Yaskawa INFORM job: OK_R2_O57-69(1)(90,0)OLD.JBI

/JOB
//NAME OK_R2_O57-69(1)(90,0)OLD
//POS
///NPOS 677,677,677,19,0,0
///TOOL 0
///POSTYPE PULSE
///PULSE
C00000=-115282,71817,32941,48127,54711,-22306
C00001=-113844,78377,40832,48113,52960,-22533
C00002=-113286,81152,44222,48167,52223,-22657
C00003=-112658,81907,45149,47913,51773,-22558
C00004=-113286,81152,44222,48167,52223,-22657
C00005=-114841,82290,45172,49039,53033,-23084
C00006=-115003,85006,48527,49507,52672,-23414
C00007=-114841,82290,45172,49039,53033,-23084
C00008=-115410,79539,41800,48987,53774,-22957
C00009=-116878,73048,33960,49005,55537,-22725
C00010=-114631,73287,21777,30026,68466,-13972
C00011=-107687,96017,31887,4043,95712,-4008
C00012=-107423,99778,39901,3942,92708,-4025
C00013=-107321,101469,43344,3906,91457,-4032
C00014=-107321,100752,43692,3904,90875,-4050
C00015=-107321,101469,43344,3906,91457,-4032
C00016=-107333,102312,44062,3909,91449,-4036
C00017=-107226,104962,47560,3875,90654,-4028
C00018=-107333,102312,44062,3909,91449,-4036
C00019=-107436,100611,40601,3946,92706,-4028
C00020=-107700,96832,32553,4047,95722,-4011
C00021=-108294,85696,32273,9932,91830,-10529
C00022=-107637,89717,40349,9733,88894,-10552
C00023=-107381,91513,43820,9663,87669,-10565
C00024=-107382,91052,44496,9665,87024,-10615
C00025=-107381,91513,43820,9663,87669,-10565
C00026=-107317,92116,44380,9645,87627,-10547
C00027=-107050,94613,47567,9574,86928,-10515
C00028=-107317,92116,44380,9645,87627,-10547
C00029=-107572,90309,40892,9715,88857,-10534
C00030=-108227,86267,32782,9914,91803,-10510
C00031=-112253,73171,16618,11071,95439,-11452
C00032=-122495,9844,5157,25727,54942,-17539
C00033=-121156,16110,12600,25480,53295,-17364
C00034=-120642,18694,15712,25408,52605,-17310
C00035=-120643,19132,17389,25673,51873,-17507
C00036=-120642,18694,15712,25408,52605,-17310
C00037=-120849,18005,15099,25505,52689,-17383
C00038=-120429,19971,16941,25331,52448,-17252
C00039=-120849,18005,15099,25505,52689,-17383
C00040=-121367,15431,12007,25581,53375,-17439
C00041=-122717,9186,4605,25835,55013,-17621
C00042=-138494,21467,-20962,-13510,88545,-918
C00043=-172227,55679,50190,-52098,32064,25809
C00044=-172226,58151,57267,-56252,30204,27980
C00045=-172259,73719,75605,-61261,28412,30549
C00046=-172259,73719,75605,-61261,28412,30549
C00047=-172291,75568,77861,-61964,28174,30905
C00048=-172279,67127,67655,-59517,29872,29717
C00049=-172279,67127,67655,-59517,29872,29717
C00050=-172707,68806,69649,-59823,29417,29854
C00051=-172279,67127,67655,-59517,29872,29717
C00052=-172484,58153,57400,-56260,30062,27978
C00053=-173076,56772,55516,-55150,29916,27380
C00054=-172487,71730,32634,-35509,46109,16330
C00055=-172505,79305,41756,-36484,44696,16958
C00056=-171934,80372,43058,-38467,45492,17923
C00057=-171699,86165,50208,-39533,44475,18576
C00058=-171934,80372,43058,-38467,45492,17923
C00059=-171934,80372,43058,-38467,45492,17923
C00060=-171934,80372,43058,-38467,45492,17923
C00061=-171934,80372,43058,-38467,45492,17923
C00062=-171934,80372,43058,-38467,45492,17923
C00063=-172992,69880,30345,-34862,46288,15983
C00064=-172199,59331,16615,-33939,49113,15228
C00065=-172399,68292,26984,-34663,47555,15757
C00066=-172399,68292,26984,-34663,47555,15757
C00067=-172079,70977,30156,-35213,47204,16071
C00068=-172399,68292,26984,-34663,47555,15757
C00069=-172399,68292,26984,-34663,47555,15757
C00070=-173084,68902,27700,-34193,47184,15559
C00071=-172399,68292,26984,-34663,47555,15757
C00072=-172399,68292,26984,-34663,47555,15757
C00073=-173171,57722,14227,-32886,49296,14681
C00074=-136545,44574,15947,-43124,46451,20365
C00075=-172050,-124043,-93312,-19428,16171,9287
C00076=-155648,-70131,-83120,13924,61027,17443
C00077=-136290,-23516,-60153,14090,83188,29885
C00078=-136350,-23051,-59906,14078,83550,29899
C00079=-136350,-23664,-59049,14098,82729,29803
C00080=-136350,-23051,-59906,14078,83550,29899
C00081=-134790,5262,-45049,12672,103577,12599
C00082=-134622,7343,-43237,12633,103510,12643
C00083=-134790,5262,-45049,12672,103577,12599
C00084=-130650,-5709,-52245,4545,96168,15148
C00085=-131657,-5407,-52003,4830,96225,14850
C00086=-130650,-5709,-52245,4545,96168,15148
C00087=-132561,-6063,-53863,7723,97717,11875
C00088=-132436,-8720,-59337,7740,99694,12036
C00089=-132445,-1782,-62924,7952,105415,12403
C00090=-141601,37323,-23290,10329,102010,9516
C00091=-93172,55874,9388,-1843,94357,23900
C00092=-93485,56784,11787,-1769,93341,23816
C00093=-93485,56329,12545,-1767,92641,23826
C00094=-93485,56784,11787,-1769,93341,23816
C00095=-93464,57012,11403,-1775,93695,23818
C00096=-93714,59095,13766,-1718,93307,23745
C00097=-93464,57012,11403,-1775,93695,23818
C00098=-94351,55649,10247,-1575,93690,23540
C00099=-95033,54913,9421,-1421,93808,23324
C00100=-94351,55649,10247,-1575,93690,23540
C00101=-94041,54751,7862,-1648,94701,23624
C00102=-93250,52756,2164,-1838,97197,23834
C00103=-93258,57323,-1415,-1867,101744,23764
C00104=-108708,74058,35602,41753,92549,11625
C00105=-107609,77867,43172,41468,89995,11080
C00106=-107179,79572,46434,41382,88936,10847
C00107=-107179,79487,47575,41378,88368,10623
C00108=-107179,79572,46434,41382,88936,10847
C00109=-85041,17756,-8276,-11251,50625,9461
C00110=-85416,19690,-6470,-10982,50459,9320
C00111=-85041,17756,-8276,-11251,50625,9461
C00112=-87036,75660,30192,-3211,91902,25887
C00113=-87645,74633,28952,-3076,92115,25688
C00114=-87036,75660,30192,-3211,91902,25887
C00115=-86708,74680,27642,-3289,92979,25963
C00116=-85872,72543,21626,-3493,95611,26155
C00117=-85876,74587,19798,-3512,97782,26092
C00118=-86821,26768,-33196,-3418,105774,25582
C00119=-56288,-65443,-100505,-9939,102051,34984
C00120=-94872,-76247,-37251,-15619,10327,-42827
C00121=-113351,-68967,-59155,816,27582,-73246
C00122=-112415,-66495,-57032,-529,27544,-72574
C00123=-112416,-66088,-55565,-540,26850,-72568
C00124=-112415,-66495,-57032,-529,27544,-72574
C00125=-125946,-59954,-52375,33832,33505,-67413
C00126=-125801,-56324,-50419,33152,34009,-67051
C00127=-125986,-60936,-52893,34026,33366,-67517
C00128=-133343,-54797,-49167,48338,43724,-75418
C00129=-132401,-55055,-49311,47843,43188,-75129
C00130=-125164,-63316,-53721,33839,32440,-67422
C00131=-126284,-65474,-55722,34821,32994,-67941
C00132=-120687,-90156,-48971,65843,10407,33929
C00133=-163424,-29173,-12092,69684,68620,47205
C00134=-170503,-20236,-5842,69401,73657,46605
C00135=-165190,-726,9323,69215,70349,47621
C00136=-177502,-61167,-55570,67933,81710,43621
C00137=-170775,-70491,-60275,67726,76450,43734
C00138=-168988,-72616,-61292,67687,75067,43782
C00139=-168256,-73449,-61686,67672,74502,43804
C00140=-168255,-73403,-61547,67686,74477,43777
C00141=-168256,-73449,-61686,67672,74502,43804
C00142=-168129,-73592,-61753,67670,74405,43808
C00143=-166480,-73871,-61885,67549,73279,44015
C00144=-168129,-73592,-61753,67670,74405,43808
C00145=-168863,-72760,-61361,67684,74971,43786
C00146=-170655,-70639,-60347,67723,76357,43737
C00147=-176850,-62168,-56094,67907,81198,43629
C00148=-197320,-70186,-60126,68463,94301,40195
C00149=-181036,-69697,-66198,61349,79658,32659
C00150=-200540,-66438,-67217,63628,100285,-15829
C00151=-127293,-88890,-117674,21964,112183,-47373
C00152=-127884,-113870,-117586,20406,100261,-49782
C00153=-127000,-93154,-82052,19489,96345,-50169
C00154=-123343,-94047,-79271,19637,93420,-49322
C00155=-121848,-94244,-78089,19702,92278,-48969
C00156=-121839,-92557,-75577,19688,91637,-49071
C00157=-121848,-94244,-78089,19702,92278,-48969
C00158=-119969,-93354,-78147,19815,92288,-48290
C00159=-118624,-93308,-78129,19884,91973,-47856
C00160=-119969,-93354,-78147,19815,92288,-48290
C00161=-121462,-93189,-79339,19761,93422,-48643
C00162=-125120,-92380,-82146,19635,96326,-49491
C00163=-116413,-89407,-85315,-11170,94586,69972
C00164=-118284,-91858,-82643,-11111,91478,69605
C00165=-119058,-92674,-81496,-11095,90266,69446
C00166=-119076,-90876,-79147,-11092,89752,69486
C00167=-119058,-92674,-81496,-11095,90266,69446
C00168=-118796,-98042,-83265,-11090,88662,69679
C00169=-118779,-98894,-83439,-11090,88340,69713
C00170=-118796,-98042,-83265,-11090,88662,69679
C00171=-123354,-93602,-81963,-11047,89491,68033
C00172=-124901,-93499,-81921,-11022,89307,67516
C00173=-123354,-93602,-81963,-11047,89491,68033
C00174=-122534,-92869,-83147,-11066,90689,68210
C00175=-120547,-90622,-85912,-11132,93767,68620
C00176=-120571,-90661,-98380,-11386,101275,67925
C00177=-125069,-105236,-119201,46912,96955,7142
C00178=-121279,-99548,-114464,46207,95099,8000
C00179=-119841,-97303,-112552,45921,94382,8319
C00180=-119848,-96543,-111162,45886,94057,8165
C00181=-119841,-97303,-112552,45921,94382,8319
C00182=-121259,-87971,-110760,46601,97668,9229
C00183=-121257,-87068,-110229,46617,97763,9276
C00184=-121259,-87971,-110760,46601,97668,9229
C00185=-122654,-89805,-112582,46929,98462,8982
C00186=-126320,-94321,-117059,47765,100534,8329
C00187=-125132,-111985,-108710,18887,62200,-22139
C00188=-122150,-102499,-103347,17190,63051,-20837
C00189=-121052,-98905,-101202,16573,63333,-20372
C00190=-121051,-97796,-99654,16626,62964,-20427
C00191=-121052,-98905,-101202,16573,63333,-20372
C00192=-120662,-97381,-100799,16308,63770,-20159
C00193=-118649,-97310,-100773,15302,63405,-19446
C00194=-120662,-97381,-100799,16308,63770,-20159
C00195=-120717,-96579,-100674,16290,64103,-20131
C00196=-120723,-93199,-99767,16143,65237,-19969
C00197=-120717,-96579,-100674,16290,64103,-20131
C00198=-121791,-100117,-102825,16885,63842,-20577
C00199=-124704,-109452,-108202,18522,63043,-21827
C00200=-114740,-109793,-107699,-22238,66313,27441
C00201=-118303,-101714,-102676,-20552,66389,26052
C00202=-119630,-98598,-100655,-19919,66404,25543
C00203=-119639,-97485,-99100,-19970,66039,25605
C00204=-119630,-98598,-100655,-19919,66404,25543
C00205=-121461,-98371,-100392,-19110,65937,24929
C00206=-122362,-98343,-100381,-18703,65740,24620
C00207=-120869,-98346,-100801,-19339,66320,25087
C00208=-120753,-95574,-99975,-19267,67213,24978
C00209=-120759,-92226,-99069,-19116,68313,24791
C00210=-120753,-95574,-99975,-19267,67213,24978
C00211=-119475,-98647,-102011,-19875,67204,25461
C00212=-116042,-106621,-107071,-21497,67130,26779
C00213=-113894,-113482,-108593,-25442,60982,30098
C00214=-117729,-104898,-103745,-23262,61171,28471
C00215=-119152,-101582,-101788,-22448,61245,27877
C00216=-119170,-99952,-99576,-22546,60754,27973
C00217=-119152,-101582,-101788,-22448,61245,27877
C00218=-121013,-102333,-103012,-21430,61098,27156
C00219=-123141,-102270,-102988,-20324,60582,26401
C00220=-121013,-102333,-103012,-21430,61098,27156
C00221=-120862,-89775,-98642,-20835,64658,26523
C00222=-120866,-85397,-96829,-20654,65721,26323
C00223=-120862,-89775,-98642,-20835,64658,26523
C00224=-119577,-92842,-100627,-21537,64647,27018
C00225=-116128,-100765,-105545,-23412,64594,28369
C00226=-120616,-96668,-103675,-23957,64374,45643
C00227=-120616,-97077,-101536,-24254,62975,45956
C00228=-120353,-97213,-100348,-24551,62319,46212
C00229=-118869,-97129,-100639,-25236,62958,46664
C00230=-120614,-98300,-102259,-24293,62807,45995
C00231=-123308,-94059,-109732,-20810,92119,41464
C00232=-120560,-97114,-101199,-23431,86244,43216
C00233=-120636,-92458,-99001,-23404,87178,43005
C00234=-120616,-97068,-101477,-23418,86408,43164
C00235=-120616,-96536,-104145,-23405,88172,42819
C00236=-120615,-97089,-97846,-24331,46439,48575
C00237=-120614,-96205,-89198,-26458,42021,49913
C00238=-120613,-95813,-87227,-26966,41113,50220
C00239=-120147,-95634,-86429,-27555,40908,50556
C00240=-118868,-95589,-86413,-28580,41350,51125
C00241=-120611,-96965,-88121,-26990,41076,50233
C00242=-120469,-95981,-105264,-23437,89109,42688
C00243=-120355,-96765,-101896,-23463,86860,43169
C00244=-119463,-95970,-102962,-19996,114254,37918
C00245=-120616,-96568,-103294,-18987,119739,36439
C00246=-120617,-95735,-106079,-19458,121767,36056
C00247=-120683,-72727,-118704,-1403,106780,1205
C00248=-120616,-97110,-101484,23732,56591,-46685
C00249=-120615,-97329,-97421,24453,54195,-47265
C00250=-120615,-97216,-95276,24833,53043,-47558
C00251=-120317,-97140,-94459,24795,52533,-47555
C00252=-120613,-98372,-96050,24869,52935,-47585
C00253=-122362,-97116,-94396,26052,53130,-48332
C00254=-120517,-95602,-107135,23321,90071,-42137
C00255=-120393,-96024,-106061,23287,89229,-42258
C00256=-120510,-96280,-105304,23307,88709,-42400
C00257=-120617,-95942,-106325,23333,89477,-42288
C00258=-120617,-94838,-108784,23367,91395,-41914
C00259=-120619,-89077,-114974,23678,97628,-40680
C00260=-119375,-87803,-114046,-9627,73434,-76892
C00261=-119874,-91001,-111320,-9540,70103,-76790
C00262=-120074,-92022,-110137,-9508,68845,-76756
C00263=-120388,-88035,-108953,-9268,70114,-76963
C00264=-120068,-92699,-111595,-9479,69387,-76797
C00265=-120617,-92323,-109789,-9348,67950,-76861
C00266=-120617,-92636,-109412,-9435,67087,-76774
C00267=-120617,-92966,-108935,-9385,65680,-76698
C00268=-120617,-93485,-108112,-8702,63167,-76584
C00269=-120617,-93807,-107566,-7310,61334,-76551
C00270=-120617,-93899,-107425,-5913,60596,-76588
C00271=-120617,-91887,-110532,-5160,63404,-76609
C00272=-120617,-91830,-110616,-4244,63440,-76636
C00273=-120617,-91600,-110911,-2665,64017,-76695
C00274=-120618,-91126,-111456,-1065,65432,-76762
C00275=-120618,-90436,-112164,126,67515,-76814
C00276=-120618,-89799,-112749,669,69377,-76843
C00277=-120618,-88579,-113586,734,71430,-76721
C00278=-120618,-87737,-114188,674,73665,-76767
C00279=-120618,-86710,-114840,-40,76341,-76871
C00280=-120619,-85981,-115253,-1370,78289,-77032
C00281=-120619,-85769,-115356,-2649,79041,-77176
C00282=-118258,-89310,-112812,-4565,75923,-76275
C00283=-117029,-89279,-112689,-5985,75998,-75947
C00284=-115084,-89307,-112300,-8369,75681,-75412
C00285=-113300,-89514,-111627,-10775,74614,-74872
C00286=-112191,-89952,-110802,-12600,72842,-74453
C00287=-112162,-90329,-110382,-13115,71673,-74372
C00288=-116808,-91534,-110372,-11031,70029,-75758
C00289=-120074,-92022,-110137,-9508,68845,-76756
C00290=-119874,-91001,-111320,-9540,70103,-76790
C00291=-119375,-87803,-114046,-9627,73434,-76892
C00292=-120613,-96141,-86612,-20456,81391,53018
C00293=-120613,-95201,-83022,-20541,79769,53295
C00294=-121508,-95240,-81659,-19950,77874,52000
C00295=-119108,-93506,-81277,-20755,79958,53812
C00296=-120703,-96226,-83293,-20548,79408,53324
C00297=-120206,-95185,-82888,-16285,85651,57184
C00298=-120275,-93619,-78099,-16321,83579,57434
C00299=-120502,-93714,-78663,-14162,87512,64436
C00300=-120613,-94474,-80645,-13297,90613,68078
C00301=-120613,-95649,-84682,-13324,92446,67881
C00302=-120615,-97441,-93706,-13451,96957,67391
C00303=-117944,-114132,-91182,23549,57658,-33742
C00304=-120612,-94052,-79174,30375,49115,-27391
C00305=-120612,-92306,-74262,31338,47277,-28046
C00306=-120611,-91624,-72518,31687,46656,-28277
C00307=-120558,-89719,-71004,31635,46677,-28249
C00308=-120609,-92783,-73582,31657,46706,-28257
C00309=-122365,-91326,-71808,32798,47083,-29054
C00310=-121100,-96285,-86968,23801,78483,-44635
C00311=-121303,-91870,-73161,24426,72832,-45883
C00312=-121523,-93334,-74795,23462,83796,-58035
C00313=-120612,-93040,-76284,23523,87550,-60648
C00314=-120612,-94304,-79928,23524,89017,-60360
C00315=-192979,-49879,-84133,31949,90821,-59300
C00316=-226136,-49296,-77583,43048,96139,-60221
C00317=-194231,-43574,-37464,64429,96533,35524
C00318=-168190,-921,2356,69742,86936,65420
C00319=-157686,-14873,-8721,69811,79682,66593
C00320=-155170,-17431,-10634,69793,77924,66853
C00321=-154140,-18406,-11354,69782,77205,66960
C00322=-154960,-19735,-12328,69815,77730,66818
C00323=-154139,-18877,-12975,69638,77486,67291
C00324=-152416,-19959,-12491,68149,70274,62953
C00325=-151462,-20771,-13080,67326,65877,57651
C00326=-150584,-21490,-13598,66880,61935,51327
C00327=-149448,-22378,-14235,66195,57985,45258
C00328=-150364,-21665,-13724,66599,59939,44567
C00329=-146294,-24621,-15825,64622,49633,44461
C00330=-147024,-24129,-15478,65026,50858,44122
C00331=-148183,-23314,-14902,65711,53127,43519
C00332=-150746,-21357,-13503,66515,56405,42739
C00333=-151844,-20450,-12847,67017,58691,42205
C00334=-154160,-18394,-11345,67568,61790,41547
C00335=-155150,-17454,-10651,67918,63984,41080
C00336=-156307,-16307,-9798,68285,66690,40524
C00337=-158578,-13896,-7981,68632,70174,39857
C00338=-158236,-14274,-8267,68563,69306,40027
C00339=-158768,-13688,-7823,68593,69674,39964
C00340=-160083,-12191,-6676,68663,70584,39811
C00341=-163356,-38025,-17867,70039,68206,46757
C00342=-171321,-47804,-23743,70196,73038,45095
C00343=-120855,-117042,-83065,287,50429,-281
C00344=-120852,-56541,-79529,233,79340,-219
C00345=-120696,51333,26745,175,69370,-180
C00346=-120686,107948,75662,172,68359,-178
C00347=-120686,108277,78684,174,66668,-180
C00348=-120673,108876,79912,172,66223,-177
C00349=-120685,108330,78544,174,66782,-180
C00350=-120704,104314,74519,181,67195,-186
C00351=-120673,108876,79912,172,66223,-177
C00352=-121521,109835,81177,5465,66399,-4971
C00353=-123474,116640,90211,14625,67368,-13734
C00354=-120128,113257,88761,29498,73318,-26772
C00355=-120686,108838,82574,29428,74862,-26590
C00356=-121763,107966,77633,29394,77512,-26324
C00357=-120686,107962,76375,6322,66410,-5366
C00358=-120686,108055,77304,6346,65890,-5395
C00359=-117369,97126,64252,10958,70846,-6903
C00360=-120686,108293,79018,6392,64962,-5445
C00361=-120992,104893,75799,6510,65219,-5544
C00362=-117369,97126,64252,10958,70846,-6903
C00363=-120630,108400,78956,19693,72345,-15662
C00364=-120761,107752,79258,26649,76197,-23334
C00365=-121775,107524,77536,26798,77367,-23449
C00366=-120025,79294,29666,22432,87187,-16596
C00367=-146832,96040,51096,-31563,98712,41471
C00368=-156862,88199,54516,-55770,96758,71489
C00369=-156858,88352,61458,-55305,94312,73083
C00370=-157852,91445,67330,-55099,92539,73648
C00371=-158245,92835,69884,-55033,91801,73892
C00372=-157951,96204,74186,-54996,91433,74294
C00373=-157784,91273,67188,-55102,92578,73662
C00374=-158040,92399,69988,-55026,91755,74041
C00375=-159291,95627,71523,-51291,93332,81554
C00376=-160209,98279,73182,-48482,94322,83905
C00377=-159956,97162,70645,-48575,95125,83623
C00378=-159321,94794,64867,-48849,97041,82959
C00379=-174197,80542,71118,-15802,102714,62389
C00380=-174195,80556,71135,-15802,102711,62390
C00381=-174195,80561,71142,-15801,102710,62390
C00382=-173773,83477,74756,-15654,102092,62625
C00383=-174194,79765,68888,-15876,103653,62265
C00384=-174199,80535,71109,-11568,105990,64366
C00385=-174198,80539,71114,-12074,105866,67869
C00386=-174201,80518,71089,-8660,108894,72599
C00387=-174202,80510,71078,-8661,108896,72599
C00388=-174205,80488,71052,-8662,108901,72597
C00389=-174210,80448,71002,-8664,108910,72595
C00390=-160796,99181,68474,-21491,79626,-54117
C00391=-160795,99200,68498,-21491,79622,-54116
C00392=-160795,99207,68507,-21491,79620,-54116
C00393=-160747,98987,66984,-21457,80402,-54239
C00394=-161332,101028,70752,-21395,79065,-54211
C00395=-160795,99207,68507,-21491,79620,-54116
C00396=-160795,99200,68498,-21491,79622,-54116
C00397=-160796,99181,68474,-21491,79626,-54117
C00398=-156887,88424,61529,-55303,94292,73080
C00399=-157880,91522,67408,-55097,92517,73646
C00400=-158273,92915,69967,-55032,91779,73890
C00401=-157979,96289,74274,-54994,91410,74293
C00402=-157812,91350,67266,-55100,92556,73660
C00403=-158068,92478,70069,-55024,91733,74039
C00404=-159318,95712,71612,-51289,93309,81552
C00405=-160236,98368,73278,-48480,94299,83903
C00406=-159983,97249,70737,-48574,95102,83621
C00407=-159349,94875,64951,-48847,97020,82956
C00408=-174197,80542,71118,-15802,102714,62389
C00409=-174195,80555,71135,-15802,102711,62390
C00410=-174195,80561,71141,-15801,102710,62390
C00411=-173773,83477,74755,-15654,102093,62624
C00412=-174194,79764,68887,-15876,103653,62265
C00413=-174199,80534,71109,-11568,105990,64366
C00414=-174198,80538,71114,-12074,105866,67869
C00415=-174201,80518,71088,-8660,108894,72599
C00416=-174202,80509,71078,-8661,108896,72599
C00417=-174205,80488,71051,-8662,108901,72597
C00418=-174210,80448,71002,-8664,108910,72595
C00419=-160796,99181,68473,-21491,79626,-54117
C00420=-160795,99199,68497,-21491,79622,-54116
C00421=-160795,99206,68506,-21491,79620,-54116
C00422=-160747,98986,66983,-21457,80402,-54239
C00423=-161332,101028,70752,-21395,79065,-54211
C00424=-160795,99206,68506,-21491,79620,-54116
C00425=-160795,99199,68497,-21491,79622,-54116
C00426=-160796,99181,68473,-21491,79626,-54117
C00427=-156915,88496,61599,-55301,94271,73077
C00428=-157907,91600,67487,-55096,92496,73644
C00429=-158301,92995,70050,-55030,91757,73888
C00430=-158006,96373,74363,-54993,91387,74291
C00431=-157840,91427,67345,-55098,92535,73658
C00432=-158096,92558,70151,-55023,91711,74037
C00433=-159346,95797,71702,-51288,93287,81550
C00434=-160263,98458,73375,-48479,94275,83902
C00435=-160010,97336,70829,-48572,95080,83619
C00436=-159376,94956,65035,-48845,96998,82954
C00437=-174197,80541,71117,-15802,102715,62389
C00438=-174195,80555,71134,-15802,102712,62390
C00439=-174195,80560,71141,-15801,102710,62390
C00440=-173773,83476,74754,-15654,102093,62624
C00441=-174194,79763,68887,-15876,103653,62265
C00442=-174199,80534,71108,-11568,105990,64366
C00443=-174198,80538,71113,-12074,105866,67869
C00444=-174201,80517,71088,-8660,108894,72599
C00445=-174203,80508,71077,-8661,108896,72599
C00446=-174205,80487,71050,-8662,108901,72597
C00447=-174210,80447,71001,-8664,108910,72595
C00448=-160796,99180,68472,-21491,79627,-54117
C00449=-160795,99198,68496,-21491,79622,-54116
C00450=-160795,99206,68506,-21491,79620,-54116
C00451=-160747,98986,66982,-21457,80402,-54239
C00452=-161332,101027,70751,-21395,79065,-54211
C00453=-160795,99206,68506,-21491,79620,-54116
C00454=-160795,99198,68496,-21491,79622,-54116
C00455=-160796,99180,68472,-21491,79627,-54117
C00456=-160394,63694,17038,-3651,83782,-73608
C00457=-190015,-23229,-64935,6709,90053,81130
C00458=-200263,9721,-38620,10181,91724,78169
C00459=-174135,-51322,-31088,61328,33879,50976
C00460=-174134,-51319,-31087,61327,33879,50977
C00461=-174133,-51978,-32760,60430,34229,51462
C00462=-175008,-52913,-31974,62066,34294,50529
C00463=-174165,-51376,-31119,68078,48326,49661
C00464=-174167,-51380,-31120,67173,48568,55955
C00465=-174192,-51426,-31146,69828,61157,64510
C00466=-174196,-51432,-31150,69829,61158,64509
C00467=-160788,-42263,-32458,15580,47921,8219
C00468=-160788,-42263,-32458,15580,47921,8219
C00469=-159909,-43388,-33874,14966,48039,8647
C00470=-161405,-44119,-33586,16024,47791,7908
C00471=-160787,-42259,-32456,15583,47920,8217
C00472=-160784,-42250,-32450,15581,47921,8219
C00473=-160783,-42246,-32448,15576,47922,8221
C00474=-160783,-42246,-32448,15576,47922,8221
C00475=-146637,-39575,-34461,6046,48590,14746
C00476=-174196,-30579,-7118,69980,41906,48750
C00477=-174191,-30568,-7111,69979,41904,48752
C00478=-174188,-30559,-7105,69977,41901,48753
C00479=-174186,-30555,-7102,69976,41901,48754
C00480=-174186,-31355,-8970,69207,42176,49221
C00481=-174962,-32094,-8117,70258,42357,48510
C00482=-174194,-30569,-7112,71825,47591,46341
C00483=-174196,-30575,-7115,70727,48120,54586
C00484=-174217,-30615,-7142,71977,59732,62495
C00485=-174219,-30621,-7146,71977,59734,62495
C00486=-174226,-30637,-7157,71978,59738,62493
C00487=-174235,-30659,-7171,71979,59742,62491
C00488=-160826,40415,13631,53464,67015,37205
C00489=-160826,40346,14725,53699,66583,36924
C00490=-160826,40419,13556,53448,67045,37224
C00491=-161205,38368,12671,53745,66948,36941
C00492=-160829,40326,14814,56358,71294,34357
C00493=-160833,40301,19018,62693,68392,39666
C00494=-160845,41308,28286,76228,74003,43895
C00495=-160845,41098,27088,76066,74172,44186
C00496=-160847,40669,24199,75673,74598,44902
C00497=-160844,40222,15431,74465,76073,47261
C00498=-107800,-52207,-58944,57218,40703,55200
C00499=-160701,2515,-37405,-57325,101772,65874
C00500=-141616,-39425,-60187,-54555,78743,60548
C00501=-117282,-83403,-80950,-58153,67097,61253
C00502=-88407,-89571,-82426,-59207,57370,57880
C00503=-68476,-97884,-84022,-50002,23247,45036
C00504=-66040,-99229,-83751,-49838,32871,-40371
C00505=-120096,-126434,-88762,51835,16555,74218
C00506=-135002,-84086,-73993,57476,43061,70498
C00507=-132040,-84680,-73570,56549,40955,71010
C00508=-131414,-81555,-71247,56056,40686,71296
C00509=-131406,-87072,-73560,57444,39877,70476
C00510=-130845,-85029,-73961,55869,40275,71397
C00511=-120653,-82966,-71266,5966,20395,75813
C00512=-120675,-82918,-71285,17010,21245,70592
C00513=-120916,-83226,-72045,25844,24084,58517
C00514=-120675,-83160,-71781,24223,23980,53145
C00515=-120675,-85948,-73873,24306,23842,53086
C00516=-120674,-86249,-74914,23862,24287,53303
C00517=-120096,-126434,-88762,51835,16555,74218
C00518=-66040,-99229,-83751,-49838,32871,-40371
C00519=-124550,-62434,-86348,-29573,82344,852
C00520=-123235,4833,-40404,-29868,88268,-211
C00521=-160797,40338,30634,-17216,54639,-7315
C00522=-160798,40335,30631,-17216,54639,-7316
C00523=-160798,40334,30630,-17216,54639,-7316
C00524=-160254,39145,28669,-17377,55324,-7200
C00525=-161179,38217,28428,-16962,54815,-7509
C00526=-160797,40338,30635,-17214,54636,-7317
C00527=-160796,40349,30645,-17215,54635,-7316
C00528=-160795,40353,30650,-17218,54637,-7314
C00529=-160795,40355,30652,-17218,54637,-7314
C00530=-160794,40358,30655,-17219,54637,-7314
C00531=-134055,6389,-12297,-27269,70214,305
C00532=-134055,6386,-12300,-27269,70214,304
C00533=-134056,6385,-12301,-27269,70214,304
C00534=-133336,6111,-13253,-27465,70843,431
C00535=-134209,4258,-14137,-27207,70198,248
C00536=-134055,6389,-12297,-27268,70211,304
C00537=-134055,6399,-12288,-27268,70211,304
C00538=-134055,6404,-12285,-27269,70214,305
C00539=-134054,6405,-12283,-27269,70214,305
C00540=-134054,6409,-12280,-27270,70214,305
C00541=-134054,6381,-12304,-27269,70214,305
C00542=-119539,-9199,-48147,-18888,87317,-2502
C00543=-107301,108516,67172,6763,80833,-7485
C00544=-107302,108543,67208,6764,80825,-7486
C00545=-107327,109506,67997,6770,80840,-7493
C00546=-107408,105168,62770,6780,81824,-7467
C00547=-107302,108837,66349,6754,81501,-7449
C00548=-107328,109508,67926,-800,79826,-3221
C00549=-107341,109965,68562,-800,79668,-3221
C00550=-107302,108679,66764,-810,80107,-3211
C00551=-107301,108507,67161,-810,79773,-3209
C00552=-107300,108486,67133,-811,79779,-3209
C00553=-105402,102050,58700,13511,85573,-11199
C00554=-105682,98756,55250,11826,82970,-6103
C00555=-105512,101987,60094,11805,81652,-6172
C00556=-107300,108776,66267,14003,84714,-11932
C00557=-107560,105371,63037,14063,84990,-11988
C00558=-108488,112185,71575,14237,83301,-12214
C00559=-109175,107441,63356,14450,86103,-12401
C00560=-110301,97927,47508,14733,91007,-12196
C00561=-132655,20555,-34602,20500,105579,-17250
C00562=-120395,-75677,-109491,17431,99945,-14261
C00563=-120731,-81008,-115648,-105,86416,-81801
C00564=-120675,-24649,-47159,-132,73228,-81771
C00565=-120676,-24635,-47149,-131,73230,-81771
C00566=-121160,-22605,-45707,73,73387,-81935
C00567=-120676,-24365,-48211,-131,74022,-81772
C00568=-121750,-24621,-47139,317,73232,-82133
C00569=-121153,-19553,-43498,69,73596,-81932
C00570=-120676,-24635,-47149,-131,73230,-81771
C00571=-120675,-24649,-47159,-132,73228,-81771
C00572=-86683,-40445,-63075,-13763,77736,-70672
C00573=-103499,26970,-9106,-7161,77072,-76192
C00574=-140778,108087,66612,-20508,92087,-48724
C00575=-140778,108110,66641,-20508,92080,-48723
C00576=-140777,108132,66670,-20508,92074,-48722
C00577=-140714,110759,70491,-20495,91150,-48542
C00578=-140777,108336,66063,-20521,92524,-48798
C00579=-141368,108983,68165,-20410,91478,-48827
C00580=-140562,116507,78152,-20494,89535,-48214
C00581=-140777,108132,66670,-20508,92074,-48722
C00582=-140778,108110,66641,-20508,92080,-48723
C00583=-140778,108110,66641,-20508,92080,-48723
C00584=-140777,108131,66669,-20508,92074,-48722
C00585=-140673,110989,70799,-20500,91092,-48518
C00586=-140777,108340,66048,-20521,92535,-48800
C00587=-141368,108987,68148,-20410,91489,-48829
C00588=-140464,116181,77719,-20509,89649,-48200
C00589=-140777,108131,66669,-20508,92075,-48722
C00590=-140778,108109,66640,-20508,92081,-48723
C00591=-140778,108086,66610,-20508,92087,-48724
C00592=-125618,13255,-41495,-24522,112345,-47401
C00593=-147482,65875,18307,-26968,106299,-45744
C00594=-160865,108111,66627,-28476,101259,-43958
C00595=-160864,108058,66881,-28455,101097,-43917
C00596=-161091,111560,73170,-28229,99189,-43527
C00597=-160867,111482,73064,-28240,99285,-43467
C00598=-160864,107969,67173,-28430,100897,-43867
C00599=-161682,111325,72860,-28215,99058,-43719
C00600=-160865,108044,66863,-28456,101100,-43918
C00601=-160866,108097,66609,-28477,101262,-43960
C00602=-160868,107404,70021,-43698,97330,-44642
C00603=-160870,107239,73702,-43453,95599,-43897
C00604=-160999,111882,81396,-43256,93800,-43188
C00605=-160873,111572,80985,-43267,93932,-43187
C00606=-160870,107239,74018,-43435,95456,-43836
C00607=-160735,111785,81268,-43268,93951,-43132
C00608=-160871,107223,73682,-43453,95602,-43899
C00609=-160869,107389,70003,-43699,97332,-44644
C00610=-160874,107343,69924,-43701,97348,-44653
C00611=-160876,107172,73597,-43455,95618,-43908
C00612=-160915,111871,81364,-43259,93852,-43174
C00613=-160879,111493,80863,-43269,93954,-43200
C00614=-160876,107172,73912,-43437,95475,-43847
C00615=-160897,112014,81553,-43255,93831,-43155
C00616=-160877,107157,73577,-43456,95621,-43910
C00617=-160875,107329,69906,-43702,97350,-44654
C00618=-160864,108120,66638,-19225,80465,79642
C00619=-160865,107719,68195,-19283,79364,79817
C00620=-160805,111145,74285,-19417,77501,80143
C00621=-160869,111315,74506,-19404,77437,80127
C00622=-160866,107660,68433,-19293,79196,79844
C00623=-161618,110659,73641,-19170,77450,79861
C00624=-160867,107705,68176,-19283,79367,79816
C00625=-160866,108106,66620,-19225,80469,79640
C00626=-132676,28155,-16568,-22865,92034,69453
C00627=-107269,-54012,-55491,-26708,77146,65149
C00628=-107269,-54016,-55493,-26708,77146,65149
C00629=-107520,-52592,-54689,-26632,77278,65024
C00630=-107269,-54165,-56823,-26643,77812,64995
C00631=-106026,-53627,-55551,-26961,77756,65482
C00632=-111625,-57136,-58581,-21094,74363,62456
C00633=-106957,-52501,-54638,-26754,77473,65192
C00634=-107270,-54018,-55494,-26707,77145,65149
C00635=-107269,-54013,-55492,-26709,77146,65149
C00636=-107266,-54027,-55500,-26709,77145,65150
C00637=-137027,-27755,-44621,6769,70731,76277
C00638=-136899,-26712,-39812,6817,68313,76184
C00639=-136540,-24439,-36585,6701,67471,76264
C00640=-136848,-26213,-39075,6804,68113,76191
C00641=-137900,-25740,-37501,7282,67483,75775
C00642=-136417,-21886,-34762,6642,67650,76319
C00643=-132357,34412,14097,4953,66227,77716
C00644=-131890,39340,18951,4768,65745,77864
C00645=-132156,38378,16523,4848,66758,77811
C00646=-132220,37154,11177,4789,69414,77897
C00647=-132226,38351,4088,4667,74376,78089
C00648=-143497,-18954,-38514,21083,45207,71474
C00649=-176671,-139811,-87877,67758,38624,43913
C00650=-136240,-146222,-94929,40423,15519,61887
C00651=-125315,3993,-19530,4296,42519,79792
C00652=-150763,-55048,-78749,-64187,60137,26500
C00653=-171462,72045,30027,-48493,41002,29627
C00654=-171613,78675,39070,-50305,39486,30716
C00655=-172205,81493,42517,-50474,38731,30888
C00656=-173558,81709,44650,-50581,37226,31105
C00657=-174312,79472,41911,-49423,37178,30537
C00658=-172205,81493,42517,-50474,38731,30888
C00659=-172212,90339,85459,-81205,28822,47225
C00660=-170941,72712,52581,-44369,37088,35289
C00661=-171235,71082,40934,-27263,47476,32443
C00662=-161709,-39449,-31108,-37959,49354,32657
C00663=-125692,-17579,-45729,-6567,64267,14209
C00664=-120682,108614,67309,63483,51839,-27699
C00665=-120682,108638,67340,63488,51836,-27703
C00666=-120682,108647,67352,63490,51834,-27704
C00667=-120457,105438,63131,62730,52144,-27175
C00668=-121241,110102,69274,64045,51982,-28035
C00669=-120682,108660,67370,63493,51832,-27706
C00670=-120686,108807,67564,63525,51814,-27729
C00671=-120686,108821,67582,63528,51813,-27732
C00672=-120686,108811,67569,63526,51814,-27730
C00673=-120686,108788,67539,63521,51817,-27727
C00674=-142392,7744,-2374,75487,63080,-35362
C00675=-109819,-108660,-86263,20744,34640,-7165
C00676=-10175,-108660,-86263,20744,-43522,-8659
BC00000=315867,805754,283188
BC00001=315867,805754,283188
BC00002=315867,805754,283188
BC00003=315867,805754,283188
BC00004=315867,805754,283188
BC00005=315867,805754,283188
BC00006=315867,805754,283188
BC00007=315867,805754,283188
BC00008=315867,805754,283188
BC00009=315867,805754,283188
BC00010=310537,817455,211903
BC00011=299248,842238,60926
BC00012=299248,842238,60926
BC00013=299248,842238,60926
BC00014=299248,842238,60926
BC00015=299248,842238,60926
BC00016=299248,842238,60926
BC00017=299248,842238,60926
BC00018=299248,842238,60926
BC00019=299248,842238,60926
BC00020=299248,842238,60926
BC00021=309010,841055,145198
BC00022=309010,841055,145198
BC00023=309010,841055,145198
BC00024=309010,841055,145198
BC00025=309010,841055,145198
BC00026=309010,841055,145198
BC00027=309010,841055,145198
BC00028=309010,841055,145198
BC00029=309010,841055,145198
BC00030=309010,841055,145198
BC00031=309010,841055,145198
BC00032=269464,830101,202581
BC00033=269464,830101,202581
BC00034=269464,830101,202581
BC00035=269464,830101,202581
BC00036=269464,830101,202581
BC00037=269464,830101,202581
BC00038=269464,830101,202581
BC00039=269464,830101,202581
BC00040=269464,830101,202581
BC00041=269464,830101,202581
BC00042=302810,780106,176804
BC00043=344903,848266,144266
BC00044=344903,848266,144266
BC00045=344903,848266,144266
BC00046=344903,848266,144266
BC00047=344903,848266,144266
BC00048=344903,848266,144261
BC00049=344903,848266,144261
BC00050=344903,848266,144261
BC00051=344903,848266,144261
BC00052=344903,848266,144265
BC00053=344903,848266,144266
BC00054=355886,834702,162552
BC00055=355886,834702,162552
BC00056=355886,834702,162552
BC00057=355886,834702,162552
BC00058=355886,834702,162552
BC00059=355886,834702,162552
BC00060=355886,834702,162552
BC00061=355886,834702,162552
BC00062=355886,834702,162552
BC00063=355886,834702,162552
BC00064=348377,844348,399871
BC00065=348377,844348,399871
BC00066=348377,844348,399871
BC00067=348377,844348,399871
BC00068=348377,844348,399871
BC00069=348377,844348,399871
BC00070=348377,844348,399871
BC00071=348377,844348,399871
BC00072=348377,844348,399871
BC00073=348377,844348,399871
BC00074=348377,717029,399871
BC00075=348377,717029,399871
BC00076=250406,701849,108605
BC00077=215945,696509,6155
BC00078=216013,696520,6358
BC00079=216013,696520,6358
BC00080=216013,696520,6358
BC00081=213892,696192,53
BC00082=213892,696192,53
BC00083=213892,696192,53
BC00084=213892,696192,53
BC00085=213892,696192,53
BC00086=213892,696192,53
BC00087=213892,696192,53
BC00088=213892,696192,53
BC00089=213892,696192,53
BC00090=227277,681725,16932
BC00091=99554,684314,33740
BC00092=99554,684314,33740
BC00093=99554,684314,33740
BC00094=99554,684314,33740
BC00095=99554,684314,33740
BC00096=99554,684314,33740
BC00097=99554,684314,33740
BC00098=99554,684314,33740
BC00099=99554,684314,33740
BC00100=99554,684314,33740
BC00101=99554,684314,33740
BC00102=99554,684314,33740
BC00103=99554,684314,33740
BC00104=69020,711056,11217
BC00105=69020,711056,11217
BC00106=69020,711056,11217
BC00107=69020,711056,11217
BC00108=69020,711056,11217
BC00109=69020,711056,11217
BC00110=69020,711056,11217
BC00111=69020,711056,11217
BC00112=69020,711056,11217
BC00113=69020,711056,11217
BC00114=69020,711056,11217
BC00115=69020,711056,11217
BC00116=69020,711056,11217
BC00117=69020,711056,11217
BC00118=69020,711056,11217
BC00119=69020,711056,11217
BC00120=224,677200,247480
BC00121=7166,683025,94113
BC00122=7166,683025,94113
BC00123=7166,683025,94113
BC00124=7166,683025,94113
BC00125=7166,683025,94113
BC00126=7165,683025,94111
BC00127=7166,683025,94113
BC00128=7166,683025,94113
BC00129=7166,683025,94113
BC00130=7166,683025,94113
BC00131=7166,683025,94113
BC00132=1273,683756,232707
BC00133=15,671225,229408
BC00134=15,671225,229408
BC00135=15,671225,229408
BC00136=15,740768,89927
BC00137=15,740768,89927
BC00138=15,744982,70925
BC00139=15,746667,63325
BC00140=15,746669,55259
BC00141=15,746667,63325
BC00142=15,747562,63916
BC00143=15,749347,63919
BC00144=15,747562,63916
BC00145=15,745877,71517
BC00146=15,741663,90519
BC00147=15,741663,90519
BC00148=15,741663,90519
BC00149=4579,733665,218396
BC00150=80822,696048,563603
BC00151=35157,680076,1075175
BC00152=35157,770360,1075175
BC00153=35157,771590,1075175
BC00154=35157,771590,1075175
BC00155=35157,771590,1075175
BC00156=35157,771590,1075175
BC00157=35157,771590,1075175
BC00158=35157,771590,1075175
BC00159=35157,771590,1075174
BC00160=35157,771590,1075175
BC00161=35157,771590,1075175
BC00162=35157,771590,1075175
BC00163=42268,766384,1075175
BC00164=42268,766384,1075175
BC00165=42268,766384,1075175
BC00166=42268,766384,1075175
BC00167=42268,766384,1075175
BC00168=42268,766384,1075175
BC00169=42268,766384,1075175
BC00170=42268,766384,1075175
BC00171=42268,766384,1075175
BC00172=42268,766384,1075175
BC00173=42268,766384,1075175
BC00174=42268,766384,1075175
BC00175=42268,766384,1075175
BC00176=42268,766384,1075175
BC00177=298709,942704,1075175
BC00178=298709,942704,1075175
BC00179=298709,942704,1075175
BC00180=298709,942704,1075175
BC00181=298709,942704,1075175
BC00182=298709,942704,1075175
BC00183=298709,942704,1075175
BC00184=298709,942704,1075175
BC00185=298709,942704,1075175
BC00186=298709,942704,1075175
BC00187=146550,860437,1075175
BC00188=146550,860437,1075175
BC00189=146550,860437,1075175
BC00190=146550,860437,1075175
BC00191=146550,860437,1075175
BC00192=146550,860437,1075175
BC00193=146550,860437,1075175
BC00194=146550,860437,1075175
BC00195=146550,860437,1075175
BC00196=146550,860437,1075175
BC00197=146550,860437,1075175
BC00198=146550,860437,1075175
BC00199=146550,860437,1075175
BC00200=175516,858216,1075175
BC00201=175516,858216,1075175
BC00202=175516,858216,1075175
BC00203=175516,858216,1075175
BC00204=175516,858216,1075175
BC00205=175516,858216,1075175
BC00206=175516,858216,1075175
BC00207=175516,858216,1075175
BC00208=175516,858216,1075175
BC00209=175516,858216,1075175
BC00210=175516,858216,1075175
BC00211=175516,858216,1075175
BC00212=175516,858216,1075175
BC00213=129379,842262,1075175
BC00214=129379,842262,1075175
BC00215=129379,842262,1075175
BC00216=129379,842262,1075175
BC00217=129379,842262,1075175
BC00218=129379,842262,1075175
BC00219=129379,842262,1075175
BC00220=129379,842262,1075175
BC00221=129379,842262,1075175
BC00222=129379,842262,1075175
BC00223=129379,842262,1075175
BC00224=129379,842262,1075175
BC00225=129379,842262,1075175
BC00226=139961,848993,1075175
BC00227=134509,852639,1075175
BC00228=132328,854097,1075175
BC00229=132328,854097,1075175
BC00230=132328,854097,1075175
BC00231=135319,889592,1075175
BC00232=135515,843339,1075175
BC00233=135533,839010,1075175
BC00234=137778,838528,1075175
BC00235=143390,837322,1075175
BC00236=181476,833990,1075175
BC00237=181497,833993,1075175
BC00238=176461,838909,1075175
BC00239=174447,840875,1075175
BC00240=174447,840875,1075175
BC00241=174447,840875,1075175
BC00242=184682,893133,1075175
BC00243=184761,874546,1075175
BC00244=174112,916325,1075175
BC00245=173642,926615,1075175
BC00246=178507,928628,1075175
BC00247=157894,860706,1075175
BC00248=129351,852868,1075175
BC00249=129362,852869,1075175
BC00250=134638,857107,1075175
BC00251=136749,858802,1075175
BC00252=136749,858802,1075175
BC00253=136749,858802,1075175
BC00254=130870,903314,1075175
BC00255=130896,897077,1075175
BC00256=130915,892748,1075175
BC00257=128672,892249,1075175
BC00258=123064,891002,1075175
BC00259=123043,890999,1075175
BC00260=398174,868421,1075175
BC00261=398174,870933,1075175
BC00262=398174,871937,1075175
BC00263=398174,871937,1075175
BC00264=398174,871937,1075175
BC00265=394352,870441,1075175
BC00266=388592,868759,1075175
BC00267=387589,867306,1075175
BC00268=385371,864886,1075175
BC00269=382181,863315,1075175
BC00270=379391,863000,1075175
BC00271=374333,882550,1075175
BC00272=372644,882866,1075175
BC00273=369951,883814,1075175
BC00274=367426,885531,1075175
BC00275=365771,887828,1075175
BC00276=365391,889807,1075175
BC00277=387166,894783,1075175
BC00278=388029,896988,1075175
BC00279=390107,899473,1075175
BC00280=393233,901117,1075175
BC00281=396017,901463,1075175
BC00282=398174,881975,1075175
BC00283=398174,881649,1075175
BC00284=398174,880650,1075175
BC00285=398174,878842,1075175
BC00286=398174,876454,1075175
BC00287=398174,875055,1075175
BC00288=398174,873339,1075175
BC00289=398174,871937,1075175
BC00290=398174,870933,1075175
BC00291=398174,868421,1075175
BC00292=48419,769941,1075175
BC00293=43349,769950,1075175
BC00294=41384,769954,1075175
BC00295=41321,769954,1075175
BC00296=41321,769954,1075175
BC00297=35772,778392,1075175
BC00298=49239,757053,1075175
BC00299=45641,763708,1075175
BC00300=44978,768291,1075175
BC00301=48083,770938,1075175
BC00302=48062,770936,1075175
BC00303=32781,783617,1075175
BC00304=28001,752077,1075175
BC00305=28012,752078,1075175
BC00306=32603,757759,1075175
BC00307=34059,759562,1075172
BC00308=34440,760032,1075175
BC00309=34440,760032,1075175
BC00310=31354,801365,1075175
BC00311=31607,741816,1075175
BC00312=33145,760208,1075171
BC00313=31586,765733,1075175
BC00314=26698,767709,1075175
BC00315=181441,722385,1075175
BC00316=206367,695978,993979
BC00317=43511,699656,343050
BC00318=15,700638,169199
BC00319=15,700638,169199
BC00320=15,702258,154627
BC00321=15,702907,148798
BC00322=15,702907,148798
BC00323=15,702907,148798
BC00324=15,695953,159545
BC00325=15,692250,164622
BC00326=15,689364,165916
BC00327=15,687048,165746
BC00328=15,688612,165744
BC00329=15,682519,161681
BC00330=15,683515,161688
BC00331=15,685058,161698
BC00332=15,689706,161726
BC00333=15,691438,161737
BC00334=15,696374,161765
BC00335=15,698216,161776
BC00336=15,700511,161790
BC00337=15,706376,161888
BC00338=15,705589,161798
BC00339=15,703851,169282
BC00340=15,699507,187994
BC00341=15,709054,229408
BC00342=15,696835,229408
BC00343=302372,698952,211490
BC00344=302372,717858,201268
BC00345=302372,750216,183774
BC00346=302372,750216,53
BC00347=302410,756221,53
BC00348=302423,758328,52
BC00349=302425,758623,53
BC00350=302425,758623,53
BC00351=302423,758328,52
BC00352=302423,758328,52
BC00353=302423,758328,52
BC00354=261483,775366,53
BC00355=261483,775366,53
BC00356=261483,775366,53
BC00357=293911,751455,53
BC00358=295135,757520,53
BC00359=272885,771858,53
BC00360=295624,759946,53
BC00361=295624,759946,53
BC00362=272885,771858,53
BC00363=277126,769514,53
BC00364=265584,778628,53
BC00365=265584,778628,53
BC00366=265584,778628,53
BC00367=355967,746549,7296
BC00368=398174,732333,10075
BC00369=398174,732336,53
BC00370=398174,726917,53
BC00371=398174,724749,53
BC00372=398174,724749,53
BC00373=398174,724749,53
BC00374=398174,724759,53
BC00375=398174,724912,53
BC00376=398174,724618,53
BC00377=398174,726661,53
BC00378=398174,731768,53
BC00379=368426,774050,236358
BC00380=368302,768625,217333
BC00381=368253,766455,209723
BC00382=368253,766455,209723
BC00383=368253,766455,209723
BC00384=361154,766186,208862
BC00385=362122,766486,208257
BC00386=355834,766353,203745
BC00387=355004,768447,211098
BC00388=352929,773681,229482
BC00389=352908,773678,283249
BC00390=390912,664927,107315
BC00391=390215,665602,80639
BC00392=389936,665872,69969
BC00393=389936,665872,69969
BC00394=389936,665872,69969
BC00395=389934,666486,69971
BC00396=390213,666216,80641
BC00397=390910,665541,107318
BC00398=398174,768127,53
BC00399=398174,762708,53
BC00400=398174,760540,53
BC00401=398174,760540,53
BC00402=398174,760540,53
BC00403=398174,760550,53
BC00404=398174,760703,53
BC00405=398174,760409,53
BC00406=398174,762452,53
BC00407=398174,767558,53
BC00408=368308,809841,236482
BC00409=368184,804416,217457
BC00410=368134,802246,209847
BC00411=368134,802246,209847
BC00412=368134,802246,209847
BC00413=361036,801977,208986
BC00414=362004,802277,208380
BC00415=355716,802144,203868
BC00416=354886,804238,211222
BC00417=352810,809472,229606
BC00418=352790,809469,283373
BC00419=390793,700718,107439
BC00420=390096,701392,80763
BC00421=389818,701662,70092
BC00422=389818,701662,70092
BC00423=389818,701662,70092
BC00424=389816,702277,70095
BC00425=390094,702007,80765
BC00426=390791,701332,107441
BC00427=398174,803918,53
BC00428=398174,798498,53
BC00429=398174,796331,53
BC00430=398174,796331,53
BC00431=398174,796331,53
BC00432=398174,796340,53
BC00433=398174,796494,53
BC00434=398174,796200,53
BC00435=398174,798243,53
BC00436=398174,803349,53
BC00437=368190,845632,236606
BC00438=368066,840207,217580
BC00439=368016,838037,209970
BC00440=368016,838037,209970
BC00441=368016,838037,209970
BC00442=360918,837768,209110
BC00443=361885,838068,208504
BC00444=355598,837935,203992
BC00445=354768,840028,211345
BC00446=352692,845263,229729
BC00447=352671,845260,283497
BC00448=390675,736509,107563
BC00449=389978,737183,80887
BC00450=389699,737453,70216
BC00451=389699,737453,70216
BC00452=389699,737453,70216
BC00453=389697,738068,70218
BC00454=389976,737798,80889
BC00455=390673,737123,107565
BC00456=390673,737123,107565
BC00457=390673,737123,107565
BC00458=390673,737123,107565
BC00459=290974,720775,160770
BC00460=290667,722939,153208
BC00461=290667,722939,153208
BC00462=290667,722939,153208
BC00463=263990,723128,151402
BC00464=263013,723888,154276
BC00465=239902,731218,144781
BC00466=238128,729410,151082
BC00467=283521,718621,232190
BC00468=282179,720936,226764
BC00469=282179,720936,226764
BC00470=282179,720936,226764
BC00471=283052,720936,222522
BC00472=284913,720944,213537
BC00473=285794,720952,209313
BC00474=287136,718637,214739
BC00475=259950,703583,235329
BC00476=279991,738060,276884
BC00477=280001,738061,250000
BC00478=280813,743470,231112
BC00479=281137,745634,223556
BC00480=281137,745634,223556
BC00481=281137,745634,223556
BC00482=273506,746410,219687
BC00483=271690,747489,222922
BC00484=250689,754377,213689
BC00485=248915,752569,219990
BC00486=244479,748048,235742
BC00487=244458,748045,289510
BC00488=271703,701029,53
BC00489=272027,703193,53
BC00490=272027,703193,53
BC00491=272027,703193,53
BC00492=266411,707508,53
BC00493=262746,705272,53
BC00494=244606,713601,53
BC00495=242832,711793,53
BC00496=238396,707272,53
BC00497=238375,707270,53
BC00498=68499,695430,53
BC00499=398174,732332,10068
BC00500=315428,722878,7554
BC00501=259600,716500,5858
BC00502=189128,708448,3717
BC00503=68499,694666,53
BC00504=15,702747,12011
BC00505=15,702747,12011
BC00506=15,702747,12011
BC00507=15,707131,53
BC00508=15,708885,53
BC00509=15,708885,53
BC00510=15,708885,53
BC00511=26435,696636,53
BC00512=12426,698694,53
BC00513=2457,701378,53
BC00514=237,702707,53
BC00515=554,700278,53
BC00516=1273,694207,10484
BC00517=15,702747,12011
BC00518=15,702747,12011
BC00519=297950,700262,21134
BC00520=297950,699644,21134
BC00521=367073,697623,223727
BC00522=363305,702964,209184
BC00523=361798,705100,203367
BC00524=361798,705100,203367
BC00525=361798,705100,203367
BC00526=362672,705098,199128
BC00527=364534,705107,190143
BC00528=365413,705116,185916
BC00529=366920,702980,191733
BC00530=370688,697639,206275
BC00531=282559,738406,156506
BC00532=278791,743746,141963
BC00533=277284,745883,136146
BC00534=277284,745883,136146
BC00535=277284,745883,136146
BC00536=278130,745881,132041
BC00537=280020,745889,122922
BC00538=280871,745899,118829
BC00539=282379,743762,124646
BC00540=286147,738422,139188
BC00541=286126,738419,192956
BC00542=298719,736844,64798
BC00543=300597,826191,171440
BC00544=303148,831060,152517
BC00545=304155,832984,145041
BC00546=304168,833008,144948
BC00547=304168,833008,144948
BC00548=314591,829616,144705
BC00549=301059,834319,144746
BC00550=296201,835994,144738
BC00551=295601,833899,152305
BC00552=294356,828576,171224
BC00553=285650,836540,171125
BC00554=290919,839813,151704
BC00555=290919,839813,151704
BC00556=290931,842229,144624
BC00557=290931,842229,144624
BC00558=309180,830430,144913
BC00559=308661,828296,152117
BC00560=308661,828296,152117
BC00561=304889,824233,171046
BC00562=304889,700105,171046
BC00563=83775,699365,9536
BC00564=83775,690394,164839
BC00565=83766,691735,138369
BC00566=83762,692272,127780
BC00567=83762,692272,127780
BC00568=83762,692272,127780
BC00569=83762,692272,127780
BC00570=83754,695342,138381
BC00571=83763,694001,164852
BC00572=83763,737347,138110
BC00573=83763,737347,138110
BC00574=197026,737412,62024
BC00575=197037,737414,35140
BC00576=197030,738091,8361
BC00577=197027,738327,1109
BC00578=197027,738361,53
BC00579=197027,738361,53
BC00580=197027,738327,1109
BC00581=197018,741702,8374
BC00582=197025,741025,35153
BC00583=196904,776946,35277
BC00584=196898,777623,8498
BC00585=196895,777893,53
BC00586=196895,777893,53
BC00587=196895,777893,53
BC00588=196895,777893,53
BC00589=196886,781207,8510
BC00590=196893,780530,35289
BC00591=196882,780528,62173
BC00592=171385,775077,62173
BC00593=195737,744422,39712
BC00594=211973,723981,24737
BC00595=211368,723652,53
BC00596=211126,723520,53
BC00597=211126,723520,53
BC00598=211126,723520,53
BC00599=211126,723520,53
BC00600=208114,721826,53
BC00601=208718,722155,24737
BC00602=205285,720250,53
BC00603=202926,718936,53
BC00604=201983,718411,53
BC00605=201983,718411,53
BC00606=201983,718411,53
BC00607=200280,717456,53
BC00608=199649,717098,53
BC00609=202008,718412,53
BC00610=190841,744312,53
BC00611=188482,742998,53
BC00612=187539,742473,53
BC00613=187539,742473,53
BC00614=187539,742473,53
BC00615=185054,741079,53
BC00616=185265,741194,53
BC00617=187624,742507,53
BC00618=211648,716653,11834
BC00619=209289,715339,53
BC00620=208346,714814,52
BC00621=208346,714814,53
BC00622=208346,714814,53
BC00623=208346,714814,52
BC00624=206012,713501,53
BC00625=208371,714815,11834
BC00626=184359,725138,114504
BC00627=162748,734429,206907
BC00628=157794,735089,185985
BC00629=155812,735353,177616
BC00630=155812,735353,177616
BC00631=155812,735353,177616
BC00632=155749,754342,177681
BC00633=155453,844081,177991
BC00634=157434,843821,186360
BC00635=162388,843161,207282
BC00636=162378,843160,234166
BC00637=147945,819524,195613
BC00638=147945,819524,195613
BC00639=147945,819524,195613
BC00640=147945,819524,195613
BC00641=147945,819524,195613
BC00642=147945,819524,195613
BC00643=147945,819524,195613
BC00644=147945,819524,195613
BC00645=147945,819524,195613
BC00646=147945,819524,195613
BC00647=147945,819524,195613
BC00648=164113,763380,121188
BC00649=164113,711732,121188
BC00650=279725,698376,121188
BC00651=279725,755875,121188
BC00652=373318,849111,338864
BC00653=359303,840797,315320
BC00654=359303,840797,315320
BC00655=359303,840797,315320
BC00656=359304,840791,337976
BC00657=359304,840791,337976
BC00658=359303,840797,315320
BC00659=359384,840891,6783
BC00660=351815,838699,3742
BC00661=350452,835380,1030
BC00662=350992,844597,341327
BC00663=342745,817956,297922
BC00664=331538,781751,238935
BC00665=337189,786996,243611
BC00666=339450,789094,245481
BC00667=339450,789094,245481
BC00668=339450,789094,245481
BC00669=339447,789098,229351
BC00670=339418,789147,54092
BC00671=339415,789152,37962
BC00672=337154,787054,36092
BC00673=331503,781810,31416
BC00674=331503,781810,310369
BC00675=331503,678865,310369
BC00676=331503,678865,310369
EC00000=798156,0
EC00001=798156,0
EC00002=798156,0
EC00003=798156,0
EC00004=798156,0
EC00005=798156,0
EC00006=798156,0
EC00007=798156,0
EC00008=798156,0
EC00009=798156,0
EC00010=798156,0
EC00011=798156,0
EC00012=798156,0
EC00013=798156,0
EC00014=798156,0
EC00015=798156,0
EC00016=798156,0
EC00017=798156,0
EC00018=798156,0
EC00019=798156,0
EC00020=798156,0
EC00021=798156,0
EC00022=798156,0
EC00023=798156,0
EC00024=798156,0
EC00025=798156,0
EC00026=798156,0
EC00027=798156,0
EC00028=798156,0
EC00029=798156,0
EC00030=798156,0
EC00031=798156,0
EC00032=798156,0
EC00033=798156,0
EC00034=798156,0
EC00035=798156,0
EC00036=798156,0
EC00037=798156,0
EC00038=798156,0
EC00039=798156,0
EC00040=798156,0
EC00041=798156,0
EC00042=798156,0
EC00043=798156,0
EC00044=798156,0
EC00045=798156,0
EC00046=798156,0
EC00047=798156,0
EC00048=798153,1
EC00049=798153,1
EC00050=798153,1
EC00051=798153,1
EC00052=798156,0
EC00053=798156,0
EC00054=798156,0
EC00055=798156,0
EC00056=798156,0
EC00057=798156,0
EC00058=798156,0
EC00059=798156,0
EC00060=798156,0
EC00061=798156,0
EC00062=798156,0
EC00063=798156,0
EC00064=798156,0
EC00065=798156,0
EC00066=798156,0
EC00067=798156,0
EC00068=798156,0
EC00069=798156,0
EC00070=798156,0
EC00071=798156,0
EC00072=798156,0
EC00073=798156,0
EC00074=798156,0
EC00075=798156,0
EC00076=798156,0
EC00077=798156,0
EC00078=798156,0
EC00079=798156,0
EC00080=798156,0
EC00081=798156,0
EC00082=798156,0
EC00083=798156,0
EC00084=798156,0
EC00085=798156,0
EC00086=798156,0
EC00087=798156,0
EC00088=798156,0
EC00089=798156,0
EC00090=798156,0
EC00091=798156,0
EC00092=798156,0
EC00093=798156,0
EC00094=798156,0
EC00095=798156,0
EC00096=798156,0
EC00097=798156,0
EC00098=798156,0
EC00099=798156,0
EC00100=798156,0
EC00101=798156,0
EC00102=798156,0
EC00103=798156,0
EC00104=798156,0
EC00105=798156,0
EC00106=798156,0
EC00107=798156,0
EC00108=798156,0
EC00109=798156,0
EC00110=798156,0
EC00111=798156,0
EC00112=798156,0
EC00113=798156,0
EC00114=798156,0
EC00115=798156,0
EC00116=798156,0
EC00117=798156,0
EC00118=798156,0
EC00119=798156,0
EC00120=798156,0
EC00121=798156,0
EC00122=798156,0
EC00123=798156,0
EC00124=798156,0
EC00125=798156,0
EC00126=798155,1
EC00127=798156,0
EC00128=798156,0
EC00129=798156,0
EC00130=798156,0
EC00131=798156,0
EC00132=798156,0
EC00133=798156,0
EC00134=798156,0
EC00135=798156,0
EC00136=798156,0
EC00137=798156,0
EC00138=798156,0
EC00139=798156,0
EC00140=798156,0
EC00141=798156,0
EC00142=798156,0
EC00143=798156,0
EC00144=798156,0
EC00145=798156,0
EC00146=798156,0
EC00147=798156,0
EC00148=798156,0
EC00149=821191,0
EC00150=883374,0
EC00151=975524,0
EC00152=975524,0
EC00153=975524,0
EC00154=975524,0
EC00155=975524,0
EC00156=975524,0
EC00157=975524,0
EC00158=975524,0
EC00159=975523,1
EC00160=975524,0
EC00161=975524,0
EC00162=975524,0
EC00163=975524,0
EC00164=975524,0
EC00165=975524,0
EC00166=975524,0
EC00167=975524,0
EC00168=975524,0
EC00169=975524,0
EC00170=975524,0
EC00171=975524,0
EC00172=975524,0
EC00173=975524,0
EC00174=975524,0
EC00175=975524,0
EC00176=975524,0
EC00177=975524,0
EC00178=975524,0
EC00179=975524,0
EC00180=975524,0
EC00181=975524,0
EC00182=975524,0
EC00183=975524,0
EC00184=975524,0
EC00185=975524,0
EC00186=975524,0
EC00187=975524,0
EC00188=975524,0
EC00189=975524,0
EC00190=975524,0
EC00191=975524,0
EC00192=975524,0
EC00193=975524,0
EC00194=975524,0
EC00195=975524,0
EC00196=975524,0
EC00197=975524,0
EC00198=975524,0
EC00199=975524,0
EC00200=975524,0
EC00201=975524,0
EC00202=975524,0
EC00203=975524,0
EC00204=975524,0
EC00205=975524,0
EC00206=975524,0
EC00207=975524,0
EC00208=975524,0
EC00209=975524,0
EC00210=975524,0
EC00211=975524,0
EC00212=975524,0
EC00213=975524,0
EC00214=975524,0
EC00215=975524,0
EC00216=975524,0
EC00217=975524,0
EC00218=975524,0
EC00219=975524,0
EC00220=975524,0
EC00221=975524,0
EC00222=975524,0
EC00223=975524,0
EC00224=975524,0
EC00225=975524,0
EC00226=975524,0
EC00227=975524,0
EC00228=975524,0
EC00229=975524,0
EC00230=975524,0
EC00231=975524,0
EC00232=975524,0
EC00233=975524,0
EC00234=975524,0
EC00235=975524,0
EC00236=975524,0
EC00237=975524,0
EC00238=975524,0
EC00239=975524,0
EC00240=975524,0
EC00241=975524,0
EC00242=975524,0
EC00243=975524,0
EC00244=975524,0
EC00245=975524,0
EC00246=975524,0
EC00247=975524,0
EC00248=975524,0
EC00249=975524,0
EC00250=975524,0
EC00251=975524,0
EC00252=975524,0
EC00253=975524,0
EC00254=975524,0
EC00255=975524,0
EC00256=975524,0
EC00257=975524,0
EC00258=975524,0
EC00259=975524,0
EC00260=975524,0
EC00261=975524,0
EC00262=975524,0
EC00263=975524,0
EC00264=975524,0
EC00265=975524,0
EC00266=975524,0
EC00267=975524,0
EC00268=975524,0
EC00269=975524,0
EC00270=975524,0
EC00271=975524,0
EC00272=975524,0
EC00273=975524,0
EC00274=975524,0
EC00275=975524,0
EC00276=975524,0
EC00277=975524,0
EC00278=975524,0
EC00279=975524,0
EC00280=975524,0
EC00281=975524,0
EC00282=975524,0
EC00283=975524,0
EC00284=975524,0
EC00285=975524,0
EC00286=975524,0
EC00287=975524,0
EC00288=975524,0
EC00289=975524,0
EC00290=975524,0
EC00291=975524,0
EC00292=975524,0
EC00293=975524,0
EC00294=975524,0
EC00295=975524,0
EC00296=975524,0
EC00297=975524,0
EC00298=975524,0
EC00299=975524,0
EC00300=975524,0
EC00301=975524,0
EC00302=975524,0
EC00303=975524,0
EC00304=975524,0
EC00305=975524,0
EC00306=975524,0
EC00307=975521,0
EC00308=975524,0
EC00309=975524,0
EC00310=975524,0
EC00311=975524,0
EC00312=975521,1
EC00313=975524,0
EC00314=975524,0
EC00315=975524,0
EC00316=959628,0
EC00317=832192,0
EC00318=798156,0
EC00319=798156,0
EC00320=798156,0
EC00321=798156,0
EC00322=798156,0
EC00323=798156,0
EC00324=798156,0
EC00325=798156,0
EC00326=798156,0
EC00327=798156,0
EC00328=798156,0
EC00329=798156,0
EC00330=798156,0
EC00331=798156,0
EC00332=798156,0
EC00333=798156,0
EC00334=798156,0
EC00335=798156,0
EC00336=798156,0
EC00337=798156,0
EC00338=798156,0
EC00339=798156,0
EC00340=798156,0
EC00341=798156,0
EC00342=798156,0
EC00343=798156,0
EC00344=798156,0
EC00345=798156,0
EC00346=798156,0
EC00347=798156,0
EC00348=798156,0
EC00349=798156,0
EC00350=798156,0
EC00351=798156,0
EC00352=798156,0
EC00353=798156,0
EC00354=798156,0
EC00355=798156,0
EC00356=798156,0
EC00357=798156,0
EC00358=798156,0
EC00359=798156,0
EC00360=798156,0
EC00361=798156,0
EC00362=798156,0
EC00363=798156,0
EC00364=798156,0
EC00365=798156,0
EC00366=798156,0
EC00367=798156,0
EC00368=798156,0
EC00369=798156,0
EC00370=798156,0
EC00371=798156,0
EC00372=798156,0
EC00373=798156,0
EC00374=798156,0
EC00375=798156,0
EC00376=798156,0
EC00377=798156,0
EC00378=798156,0
EC00379=798156,0
EC00380=798156,0
EC00381=798156,0
EC00382=798156,0
EC00383=798156,0
EC00384=798156,0
EC00385=798156,0
EC00386=798156,0
EC00387=798156,0
EC00388=798156,0
EC00389=798156,0
EC00390=798156,0
EC00391=798156,0
EC00392=798156,0
EC00393=798156,0
EC00394=798156,0
EC00395=798156,0
EC00396=798156,0
EC00397=798156,0
EC00398=798156,0
EC00399=798156,0
EC00400=798156,0
EC00401=798156,0
EC00402=798156,0
EC00403=798156,0
EC00404=798156,0
EC00405=798156,0
EC00406=798156,0
EC00407=798156,0
EC00408=798156,0
EC00409=798156,0
EC00410=798156,0
EC00411=798156,0
EC00412=798156,0
EC00413=798156,0
EC00414=798156,0
EC00415=798156,0
EC00416=798156,0
EC00417=798156,0
EC00418=798156,0
EC00419=798156,0
EC00420=798156,0
EC00421=798156,0
EC00422=798156,0
EC00423=798156,0
EC00424=798156,0
EC00425=798156,0
EC00426=798156,0
EC00427=798156,0
EC00428=798156,0
EC00429=798156,0
EC00430=798156,0
EC00431=798156,0
EC00432=798156,0
EC00433=798156,0
EC00434=798156,0
EC00435=798156,0
EC00436=798156,0
EC00437=798156,0
EC00438=798156,0
EC00439=798156,0
EC00440=798156,0
EC00441=798156,0
EC00442=798156,0
EC00443=798156,0
EC00444=798156,0
EC00445=798156,0
EC00446=798156,0
EC00447=798156,0
EC00448=798156,0
EC00449=798156,0
EC00450=798156,0
EC00451=798156,0
EC00452=798156,0
EC00453=798156,0
EC00454=798156,0
EC00455=798156,0
EC00456=798156,0
EC00457=798156,0
EC00458=798156,0
EC00459=798156,0
EC00460=798156,0
EC00461=798156,0
EC00462=798156,0
EC00463=798156,0
EC00464=798156,0
EC00465=798156,0
EC00466=798156,0
EC00467=798156,0
EC00468=798156,0
EC00469=798156,0
EC00470=798156,0
EC00471=798156,0
EC00472=798156,0
EC00473=798156,0
EC00474=798156,0
EC00475=798156,0
EC00476=798156,0
EC00477=798156,0
EC00478=798156,0
EC00479=798156,0
EC00480=798156,0
EC00481=798156,0
EC00482=798156,0
EC00483=798156,0
EC00484=798156,0
EC00485=798156,0
EC00486=798156,0
EC00487=798156,0
EC00488=798156,0
EC00489=798156,0
EC00490=798156,0
EC00491=798156,0
EC00492=798156,0
EC00493=798156,0
EC00494=798156,0
EC00495=798156,0
EC00496=798156,0
EC00497=798156,0
EC00498=798156,0
EC00499=798153,1
EC00500=798154,1
EC00501=798154,1
EC00502=798155,1
EC00503=798156,0
EC00504=798156,0
EC00505=798156,0
EC00506=798156,0
EC00507=798156,0
EC00508=798156,0
EC00509=798156,0
EC00510=798156,0
EC00511=798156,0
EC00512=798156,0
EC00513=798156,0
EC00514=798156,0
EC00515=798156,0
EC00516=798156,0
EC00517=798156,0
EC00518=798156,0
EC00519=798156,0
EC00520=798156,0
EC00521=798156,0
EC00522=798156,0
EC00523=798156,0
EC00524=798156,0
EC00525=798156,0
EC00526=798156,0
EC00527=798156,0
EC00528=798156,0
EC00529=798156,0
EC00530=798156,0
EC00531=798156,0
EC00532=798156,0
EC00533=798156,0
EC00534=798156,0
EC00535=798156,0
EC00536=798156,0
EC00537=798156,0
EC00538=798156,0
EC00539=798156,0
EC00540=798156,0
EC00541=798156,0
EC00542=798156,0
EC00543=798156,0
EC00544=798156,0
EC00545=798156,0
EC00546=798156,0
EC00547=798156,0
EC00548=798156,0
EC00549=798156,0
EC00550=798156,0
EC00551=798156,0
EC00552=798156,0
EC00553=798156,0
EC00554=798156,0
EC00555=798156,0
EC00556=798156,0
EC00557=798156,0
EC00558=798156,0
EC00559=798156,0
EC00560=798156,0
EC00561=798156,0
EC00562=798156,0
EC00563=798156,0
EC00564=798156,0
EC00565=798156,0
EC00566=798156,0
EC00567=798156,0
EC00568=798156,0
EC00569=798156,0
EC00570=798156,0
EC00571=798156,0
EC00572=798156,0
EC00573=798156,0
EC00574=798156,0
EC00575=798156,0
EC00576=798156,0
EC00577=798156,0
EC00578=798156,0
EC00579=798156,0
EC00580=798156,0
EC00581=798156,0
EC00582=798156,0
EC00583=798156,0
EC00584=798156,0
EC00585=798156,0
EC00586=798156,0
EC00587=798156,0
EC00588=798156,0
EC00589=798156,0
EC00590=798156,0
EC00591=798156,0
EC00592=798156,0
EC00593=798156,0
EC00594=798156,0
EC00595=798156,0
EC00596=798156,0
EC00597=798156,0
EC00598=798156,0
EC00599=798156,0
EC00600=798156,0
EC00601=798156,0
EC00602=798156,0
EC00603=798156,0
EC00604=798156,0
EC00605=798156,0
EC00606=798156,0
EC00607=798156,0
EC00608=798156,0
EC00609=798156,0
EC00610=798156,0
EC00611=798156,0
EC00612=798156,0
EC00613=798156,0
EC00614=798156,0
EC00615=798156,0
EC00616=798156,0
EC00617=798156,0
EC00618=798156,0
EC00619=798156,0
EC00620=798155,0
EC00621=798156,0
EC00622=798156,0
EC00623=798155,0
EC00624=798156,0
EC00625=798156,0
EC00626=798156,0
EC00627=798156,0
EC00628=798156,0
EC00629=798156,0
EC00630=798156,0
EC00631=798156,0
EC00632=798156,0
EC00633=798156,0
EC00634=798156,0
EC00635=798156,0
EC00636=798156,0
EC00637=798156,0
EC00638=798156,0
EC00639=798156,0
EC00640=798156,0
EC00641=798156,0
EC00642=798156,0
EC00643=798156,0
EC00644=798156,0
EC00645=798156,0
EC00646=798156,0
EC00647=798156,0
EC00648=798156,0
EC00649=798156,0
EC00650=798156,0
EC00651=798156,0
EC00652=798156,0
EC00653=798155,1
EC00654=798155,1
EC00655=798155,1
EC00656=798156,0
EC00657=798156,0
EC00658=798155,1
EC00659=798155,1
EC00660=798155,1
EC00661=798156,0
EC00662=798156,0
EC00663=798156,0
EC00664=798156,0
EC00665=798156,0
EC00666=798156,0
EC00667=798156,0
EC00668=798156,0
EC00669=798156,0
EC00670=798156,0
EC00671=798156,0
EC00672=798156,0
EC00673=798156,0
EC00674=798156,0
EC00675=798156,0
EC00676=798156,0
///POSTYPE BASE
///RECTAN
///RCONF 0,0,0,0,0,0,0,0,0,0,0,0,0,0,0,0,0,0,0,0,0,0,0,0
P00006=0.222,-3.123,-1.508,0.0000,0.0000,0.0000
P00021=-0.225,-6.128,-0.405,0.0000,0.0000,0.0000
P00022=0.222,-3.123,-1.508,0.0000,0.0000,0.0000
P00023=0.143,-0.036,0.682,0.0000,0.0000,0.0000
P00024=0.145,-0.552,1.326,0.0000,0.0000,0.0000
P00025=-2.003,0.006,0.728,0.0000,0.0000,0.0000
P00026=0.562,-0.002,-0.337,0.0000,0.0000,0.0000
P00027=-0.746,0.015,-9.096,0.0000,0.0000,0.0000
P00028=-2.237,-0.018,-7.702,0.0000,0.0000,0.0000
P00029=-2.156,-0.086,-4.681,0.0000,0.0000,0.0000
P00030=5.926,-4.294,-1.390,0.0000,0.0000,0.0000
P00031=1.853,-0.001,-1.549,0.0000,0.0000,0.0000
P00032=1.957,0.503,-7.217,0.0000,0.0000,0.0000
P00041=0.192,3.924,0.305,0.0000,0.0000,0.0000
P00042=-0.217,1.941,0.413,0.0000,0.0000,0.0000
P00043=-0.044,-1.937,1.197,0.0000,0.0000,0.0000
P00044=0.687,-2.322,1.156,0.0000,0.0000,0.0000
P00045=-0.068,-0.810,1.603,0.0000,0.0000,0.0000
P00046=0.799,0.043,1.292,0.0000,0.0000,0.0000
//INST
///DATE 2024/01/08 17:07
///ATTR SC,RW
///GROUP1 RB1,BS1
///GROUP2 ST1
NOP
'OK_r2_O57-69(1)(90,0)
'Down
'Path S1900
SFTOF3D
MOVJ C00000 BC00000 VJ=100.00  +MOVJ EC00000 VJ=100.00
MOVL C00001 BC00001 V=100.0  +MOVJ EC00001 VJ=100.00
SMOVL C00002 BC00002 V=60.0  +MOVJ EC00002
SREFP 3 C00003 BC00003  +REFP EC00003
CALL JOB:SEARCH-R1-S13D
SET P031 P006
SFTON3D P031
SMOVL C00004 BC00004 V=60.0  +MOVJ EC00004
SMOVL C00005 BC00005 V=60.0  +MOVJ EC00005
SREFP 3 C00006 BC00006  +REFP EC00006
CALL JOB:SEARCH-R1-S13D
SET P031 P006
SFTON3D P031
SMOVL C00007 BC00007 V=60.0  +MOVJ EC00007
MOVL C00008 BC00008 V=400.0  +MOVJ EC00008 VJ=100.00
MOVL C00009 BC00009 V=1000.0  +MOVJ EC00009 VJ=100.00
'Path S1901
SFTOF3D
PAUSE
MOVJ C00010 BC00010 VJ=100.00  +MOVJ EC00010 VJ=100.00
MOVJ C00011 BC00011 VJ=100.00  +MOVJ EC00011 VJ=100.00
MOVL C00012 BC00012 V=100.0  +MOVJ EC00012 VJ=100.00
SMOVL C00013 BC00013 V=60.0  +MOVJ EC00013
SREFP 3 C00014 BC00014  +REFP EC00014
CALL JOB:SEARCH-R1-S13D
SET P026 P006
SFTON3D P026
SMOVL C00015 BC00015 V=60.0  +MOVJ EC00015
SMOVL C00016 BC00016 V=60.0  +MOVJ EC00016
SREFP 3 C00017 BC00017  +REFP EC00017
CALL JOB:SEARCH-R1-S13D
SET P026 P006
SFTON3D P026
SMOVL C00018 BC00018 V=60.0  +MOVJ EC00018
MOVL C00019 BC00019 V=400.0  +MOVJ EC00019 VJ=100.00
MOVL C00020 BC00020 V=1000.0  +MOVJ EC00020 VJ=100.00
'Path S1902
SFTOF3D
MOVJ C00021 BC00021 VJ=100.00  +MOVJ EC00021 VJ=100.00
MOVL C00022 BC00022 V=100.0  +MOVJ EC00022 VJ=100.00
SMOVL C00023 BC00023 V=60.0  +MOVJ EC00023
SREFP 3 C00024 BC00024  +REFP EC00024
CALL JOB:SEARCH-R1-S13D
SET P027 P006
SFTON3D P027
SMOVL C00025 BC00025 V=60.0  +MOVJ EC00025
SMOVL C00026 BC00026 V=60.0  +MOVJ EC00026
SREFP 3 C00027 BC00027  +REFP EC00027
CALL JOB:SEARCH-R1-S13D
SET P027 P006
SFTON3D P027
SMOVL C00028 BC00028 V=60.0  +MOVJ EC00028
MOVL C00029 BC00029 V=400.0  +MOVJ EC00029 VJ=100.00
MOVL C00030 BC00030 V=1000.0  +MOVJ EC00030 VJ=100.00
'Path S1903
SFTOF3D
SMOVL C00031 BC00031 V=83.3  +MOVJ EC00031
MOVJ C00032 BC00032 VJ=100.00  +MOVJ EC00032 VJ=100.00
MOVL C00033 BC00033 V=100.0  +MOVJ EC00033 VJ=100.00
SMOVL C00034 BC00034 V=60.0  +MOVJ EC00034
SREFP 3 C00035 BC00035  +REFP EC00035
CALL JOB:SEARCH-R1-S13D
SET P022 P006
SFTON3D P022
SMOVL C00036 BC00036 V=60.0  +MOVJ EC00036
SMOVL C00037 BC00037 V=60.0  +MOVJ EC00037
SREFP 3 C00038 BC00038  +REFP EC00038
CALL JOB:SEARCH-R1-S13D
SET P022 P006
SFTON3D P022
SMOVL C00039 BC00039 V=60.0  +MOVJ EC00039
MOVL C00040 BC00040 V=400.0  +MOVJ EC00040 VJ=100.00
MOVL C00041 BC00041 V=1000.0  +MOVJ EC00041 VJ=100.00
MOVJ C00042 BC00042 VJ=100.00  +MOVJ EC00042 VJ=100.00
'Path S1904
SFTOF3D
MOVJ C00043 BC00043 VJ=100.00  +MOVJ EC00043 VJ=100.00
MOVJ C00044 BC00044 VJ=100.00  +MOVJ EC00044 VJ=100.00
MOVL C00045 BC00045 V=400.0  +MOVJ EC00045 VJ=100.00
SMOVL C00046 BC00046 V=60.0  +MOVJ EC00046
SREFP 3 C00047 BC00047  +REFP EC00047
CALL JOB:SEARCH-R1-S13D
SET P028 P006
SFTON3D P028
SMOVL C00048 BC00048 V=60.0  +MOVJ EC00048
SMOVL C00049 BC00049 V=60.0  +MOVJ EC00049
SREFP 3 C00050 BC00050  +REFP EC00050
CALL JOB:SEARCH-R1-S13D
SET P028 P006
SFTON3D P028
SMOVL C00051 BC00051 V=60.0  +MOVJ EC00051
MOVL C00052 BC00052 V=400.0  +MOVJ EC00052 VJ=100.00
MOVL C00053 BC00053 V=1000.0  +MOVJ EC00053 VJ=100.00
'Path S1905
SFTOF3D
MOVJ C00054 BC00054 VJ=100.00  +MOVJ EC00054 VJ=100.00
MOVL C00055 BC00055 V=100.0  +MOVJ EC00055 VJ=100.00
SMOVL C00056 BC00056 V=60.0  +MOVJ EC00056
SREFP 3 C00057 BC00057  +REFP EC00057
CALL JOB:SEARCH-R1-S13D
SET P029 P006
SFTON3D P029
SMOVL C00058 BC00058 V=60.0  +MOVJ EC00058
SMOVL C00059 BC00059 V=60.0  +MOVJ EC00059
SREFP 3 C00060 BC00060  +REFP EC00060
CALL JOB:SEARCH-R1-S13D
SET P029 P006
SFTON3D P029
SMOVL C00061 BC00061 V=60.0  +MOVJ EC00061
MOVL C00062 BC00062 V=400.0  +MOVJ EC00062 VJ=100.00
MOVL C00063 BC00063 V=1000.0  +MOVJ EC00063 VJ=100.00
'Path S1906
SFTOF3D
MOVJ C00064 BC00064 VJ=100.00  +MOVJ EC00064 VJ=100.00
MOVL C00065 BC00065 V=100.0  +MOVJ EC00065 VJ=100.00
SMOVL C00066 BC00066 V=60.0  +MOVJ EC00066
SREFP 3 C00067 BC00067  +REFP EC00067
CALL JOB:SEARCH-R1-S13D
SET P030 P006
SFTON3D P030
SMOVL C00068 BC00068 V=60.0  +MOVJ EC00068
SMOVL C00069 BC00069 V=60.0  +MOVJ EC00069
SREFP 3 C00070 BC00070  +REFP EC00070
CALL JOB:SEARCH-R1-S13D
SET P030 P006
SFTON3D P030
SMOVL C00071 BC00071 V=60.0  +MOVJ EC00071
MOVL C00072 BC00072 V=400.0  +MOVJ EC00072 VJ=100.00
MOVL C00073 BC00073 V=1000.0  +MOVJ EC00073 VJ=100.00
MOVJ C00074 BC00074 VJ=100.00  +MOVJ EC00074 VJ=100.00
MOVJ C00075 BC00075 VJ=100.00  +MOVJ EC00075 VJ=100.00
MOVJ C00076 BC00076 VJ=100.00  +MOVJ EC00076 VJ=100.00
COMM 'Path S1907
COMM SFTOF3D
COMM MOVL C00077 BC00077 V=400.0  +MOVJ EC00077 VJ=100.00
COMM SMOVL C00078 BC00078 V=60.0  +MOVJ EC00078
COMM SREFP 3 C00079 BC00079  +REFP EC00079
COMM CALL JOB:SEARCH-R1-S13D
COMM SET P023 P006
COMM SFTON3D P023
COMM SMOVL C00080 BC00080 V=60.0  +MOVJ EC00080
COMM SMOVL C00081 BC00081 V=60.0  +MOVJ EC00081
COMM SREFP 3 C00082 BC00082  +REFP EC00082
COMM CALL JOB:SEARCH-R1-S13D
COMM SET P023 P006
COMM SFTON3D P023
COMM SMOVL C00083 BC00083 V=60.0  +MOVJ EC00083
COMM SMOVL C00084 BC00084 V=60.0  +MOVJ EC00084
COMM SREFP 3 C00085 BC00085  +REFP EC00085
COMM CALL JOB:SEARCH-R1-S13D
COMM SET P023 P006
COMM SFTON3D P023
COMM SMOVL C00086 BC00086 V=60.0  +MOVJ EC00086
COMM MOVL C00087 BC00087 V=400.0  +MOVJ EC00087 VJ=100.00
COMM MOVL C00088 BC00088 V=1000.0  +MOVJ EC00088 VJ=100.00
COMM MOVL C00089 BC00089 V=1000.0  +MOVJ EC00089 VJ=100.00
COMM MOVJ C00090 BC00090 VJ=100.00  +MOVJ EC00090 VJ=100.00
COMM 'Path S1908
COMM SFTOF3D
COMM MOVL C00091 BC00091 V=400.0  +MOVJ EC00091 VJ=100.00
COMM SMOVL C00092 BC00092 V=60.0  +MOVJ EC00092
COMM SREFP 3 C00093 BC00093  +REFP EC00093
COMM CALL JOB:SEARCH-R1-S13D
COMM SET P024 P006
COMM SFTON3D P024
COMM SMOVL C00094 BC00094 V=60.0  +MOVJ EC00094
COMM SMOVL C00095 BC00095 V=60.0  +MOVJ EC00095
COMM SREFP 3 C00096 BC00096  +REFP EC00096
COMM CALL JOB:SEARCH-R1-S13D
COMM SET P024 P006
COMM SFTON3D P024
COMM SMOVL C00097 BC00097 V=60.0  +MOVJ EC00097
COMM SMOVL C00098 BC00098 V=60.0  +MOVJ EC00098
COMM SREFP 3 C00099 BC00099  +REFP EC00099
COMM CALL JOB:SEARCH-R1-S13D
COMM SET P024 P006
COMM SFTON3D P024
COMM SMOVL C00100 BC00100 V=60.0  +MOVJ EC00100
COMM MOVL C00101 BC00101 V=400.0  +MOVJ EC00101 VJ=100.00
COMM MOVL C00102 BC00102 V=1000.0  +MOVJ EC00102 VJ=100.00
COMM MOVL C00103 BC00103 V=1000.0  +MOVJ EC00103 VJ=100.00
COMM 'Path S1909
COMM SFTOF3D
COMM MOVJ C00104 BC00104 VJ=100.00  +MOVJ EC00104 VJ=100.00
COMM MOVL C00105 BC00105 V=400.0  +MOVJ EC00105 VJ=100.00
COMM SMOVL C00106 BC00106 V=60.0  +MOVJ EC00106
COMM SREFP 3 C00107 BC00107  +REFP EC00107
COMM CALL JOB:SEARCH-R1-S13D
COMM SET P025 P006
COMM SFTON3D P025
COMM SMOVL C00108 BC00108 V=60.0  +MOVJ EC00108
COMM SMOVL C00109 BC00109 V=60.0  +MOVJ EC00109
COMM SREFP 3 C00110 BC00110  +REFP EC00110
COMM CALL JOB:SEARCH-R1-S13D
COMM SET P025 P006
COMM SFTON3D P025
COMM SMOVL C00111 BC00111 V=60.0  +MOVJ EC00111
COMM SMOVL C00112 BC00112 V=60.0  +MOVJ EC00112
COMM SREFP 3 C00113 BC00113  +REFP EC00113
COMM CALL JOB:SEARCH-R1-S13D
COMM SET P025 P006
COMM SFTON3D P025
COMM SMOVL C00114 BC00114 V=60.0  +MOVJ EC00114
COMM MOVL C00115 BC00115 V=400.0  +MOVJ EC00115 VJ=100.00
COMM MOVL C00116 BC00116 V=1000.0  +MOVJ EC00116 VJ=100.00
COMM MOVL C00117 BC00117 V=1000.0  +MOVJ EC00117 VJ=100.00
COMM MOVJ C00118 BC00118 VJ=100.00  +MOVJ EC00118 VJ=100.00
MOVJ C00119 BC00119 VJ=100.00  +MOVJ EC00119 VJ=100.00
MOVJ C00120 BC00120 VJ=100.00  +MOVJ EC00120 VJ=100.00
'Path S1910
SFTOF3D
MOVL C00121 BC00121 V=100.0  +MOVJ EC00121 VJ=100.00
SMOVL C00122 BC00122 V=60.0  +MOVJ EC00122
SREFP 3 C00123 BC00123  +REFP EC00123
CALL JOB:SEARCH-R1-S13D
SET P021 P006
SFTON3D P021
SMOVL C00124 BC00124 V=60.0  +MOVJ EC00124
SMOVL C00125 BC00125 V=60.0  +MOVJ EC00125
SREFP 3 C00126 BC00126  +REFP EC00126
CALL JOB:SEARCH-R1-S13D
SET P021 P006
SFTON3D P021
SMOVL C00127 BC00127 V=60.0  +MOVJ EC00127
SMOVL C00128 BC00128 V=60.0  +MOVJ EC00128
SREFP 3 C00129 BC00129  +REFP EC00129
CALL JOB:SEARCH-R1-S13D
SET P021 P006
SFTON3D P021
SMOVL C00130 BC00130 V=60.0  +MOVJ EC00130
MOVL C00131 BC00131 V=400.0  +MOVJ EC00131 VJ=100.00
MOVJ C00132 BC00132 VJ=100.00  +MOVJ EC00132 VJ=100.00
MOVJ C00133 BC00133 VJ=100.00  +MOVJ EC00133 VJ=100.00
MOVJ C00134 BC00134 VJ=50.00  +MOVJ EC00134 VJ=50.00
MOVJ C00135 BC00135 VJ=50.00  +MOVJ EC00135 VJ=50.00
MOVJ C00136 BC00136 VJ=100.00  +MOVJ EC00136 VJ=100.00
'Path S1912
SFTOF3D
MOVJ C00137 BC00137 VJ=100.00  +MOVJ EC00137 VJ=100.00
MOVL C00138 BC00138 V=400.0  +MOVJ EC00138 VJ=100.00
SMOVL C00139 BC00139 V=60.0  +MOVJ EC00139
SREFP 3 C00140 BC00140  +REFP EC00140
CALL JOB:SEARCH-R1-S13D
SET P032 P006
SFTON3D P032
SMOVL C00141 BC00141 V=60.0  +MOVJ EC00141
SMOVL C00142 BC00142 V=60.0  +MOVJ EC00142
SREFP 3 C00143 BC00143  +REFP EC00143
CALL JOB:SEARCH-R1-S13D
SET P032 P006
SFTON3D P032
SMOVL C00144 BC00144 V=60.0  +MOVJ EC00144
MOVL C00145 BC00145 V=400.0  +MOVJ EC00145 VJ=100.00
MOVL C00146 BC00146 V=1000.0  +MOVJ EC00146 VJ=100.00
'Up
MOVJ C00147 BC00147 VJ=50.00  +MOVJ EC00147 VJ=50.00
MOVJ C00148 BC00148 VJ=50.00  +MOVJ EC00148 VJ=50.00
MOVJ C00149 BC00149 VJ=100.00  +MOVJ EC00149 VJ=100.00
MOVJ C00150 BC00150 VJ=100.00  +MOVJ EC00150 VJ=100.00
MOVJ C00151 BC00151 VJ=100.00  +MOVJ EC00151 VJ=100.00
MOVJ C00152 BC00152 VJ=100.00  +MOVJ EC00152 VJ=100.00
'Path S1137
SFTOF3D
MOVJ C00153 BC00153 VJ=100.00  +MOVJ EC00153 VJ=100.00
MOVL C00154 BC00154 V=400.0  +MOVJ EC00154 VJ=100.00
SMOVL C00155 BC00155 V=60.0  +MOVJ EC00155
SREFP 3 C00156 BC00156  +REFP EC00156
CALL JOB:SEARCH-R1-S13D
SET P046 P006
SFTON3D P046
SMOVL C00157 BC00157 V=60.0  +MOVJ EC00157
SMOVL C00158 BC00158 V=60.0  +MOVJ EC00158
SREFP 3 C00159 BC00159  +REFP EC00159
CALL JOB:SEARCH-R1-S13D
SET P046 P006
SFTON3D P046
SMOVL C00160 BC00160 V=60.0  +MOVJ EC00160
MOVL C00161 BC00161 V=400.0  +MOVJ EC00161 VJ=100.00
MOVL C00162 BC00162 V=1000.0  +MOVJ EC00162 VJ=100.00
'Path S1169
SFTOF3D
MOVJ C00163 BC00163 VJ=100.00  +MOVJ EC00163 VJ=100.00
MOVL C00164 BC00164 V=400.0  +MOVJ EC00164 VJ=100.00
SMOVL C00165 BC00165 V=60.0  +MOVJ EC00165
SREFP 3 C00166 BC00166  +REFP EC00166
CALL JOB:SEARCH-R1-S13D
SET P045 P006
SFTON3D P045
SMOVL C00167 BC00167 V=60.0  +MOVJ EC00167
SMOVL C00168 BC00168 V=60.0  +MOVJ EC00168
SREFP 3 C00169 BC00169  +REFP EC00169
CALL JOB:SEARCH-R1-S13D
SET P045 P006
SFTON3D P045
SMOVL C00170 BC00170 V=60.0  +MOVJ EC00170
SMOVL C00171 BC00171 V=60.0  +MOVJ EC00171
SREFP 3 C00172 BC00172  +REFP EC00172
CALL JOB:SEARCH-R1-S13D
SET P045 P006
SFTON3D P045
SMOVL C00173 BC00173 V=60.0  +MOVJ EC00173
MOVL C00174 BC00174 V=400.0  +MOVJ EC00174 VJ=100.00
MOVL C00175 BC00175 V=1000.0  +MOVJ EC00175 VJ=100.00
MOVL C00176 BC00176 V=1000.0  +MOVJ EC00176 VJ=100.00
'Path S1168
SFTOF3D
MOVJ C00177 BC00177 VJ=100.00  +MOVJ EC00177 VJ=100.00
MOVL C00178 BC00178 V=400.0  +MOVJ EC00178 VJ=100.00
SMOVL C00179 BC00179 V=60.0  +MOVJ EC00179
SREFP 3 C00180 BC00180  +REFP EC00180
CALL JOB:SEARCH-R1-S13D
SET P044 P006
SFTON3D P044
SMOVL C00181 BC00181 V=60.0  +MOVJ EC00181
SMOVL C00182 BC00182 V=60.0  +MOVJ EC00182
SREFP 3 C00183 BC00183  +REFP EC00183
CALL JOB:SEARCH-R1-S13D
SET P044 P006
SFTON3D P044
SMOVL C00184 BC00184 V=60.0  +MOVJ EC00184
MOVL C00185 BC00185 V=400.0  +MOVJ EC00185 VJ=100.00
MOVL C00186 BC00186 V=1000.0  +MOVJ EC00186 VJ=100.00
'Path S1167
SFTOF3D
MOVJ C00187 BC00187 VJ=100.00  +MOVJ EC00187 VJ=100.00
MOVL C00188 BC00188 V=400.0  +MOVJ EC00188 VJ=100.00
SMOVL C00189 BC00189 V=60.0  +MOVJ EC00189
SREFP 3 C00190 BC00190  +REFP EC00190
CALL JOB:SEARCH-R1-S13D
SET P043 P006
SFTON3D P043
SMOVL C00191 BC00191 V=60.0  +MOVJ EC00191
SMOVL C00192 BC00192 V=60.0  +MOVJ EC00192
SREFP 3 C00193 BC00193  +REFP EC00193
CALL JOB:SEARCH-R1-S13D
SET P043 P006
SFTON3D P043
SMOVL C00194 BC00194 V=60.0  +MOVJ EC00194
SMOVL C00195 BC00195 V=60.0  +MOVJ EC00195
SREFP 3 C00196 BC00196  +REFP EC00196
CALL JOB:SEARCH-R1-S13D
SET P043 P006
SFTON3D P043
SMOVL C00197 BC00197 V=60.0  +MOVJ EC00197
MOVL C00198 BC00198 V=400.0  +MOVJ EC00198 VJ=100.00
MOVL C00199 BC00199 V=1000.0  +MOVJ EC00199 VJ=100.00
'Path S1166
SFTOF3D
MOVJ C00200 BC00200 VJ=100.00  +MOVJ EC00200 VJ=100.00
MOVL C00201 BC00201 V=400.0  +MOVJ EC00201 VJ=100.00
SMOVL C00202 BC00202 V=60.0  +MOVJ EC00202
SREFP 3 C00203 BC00203  +REFP EC00203
CALL JOB:SEARCH-R1-S13D
SET P042 P006
SFTON3D P042
SMOVL C00204 BC00204 V=60.0  +MOVJ EC00204
SMOVL C00205 BC00205 V=60.0  +MOVJ EC00205
SREFP 3 C00206 BC00206  +REFP EC00206
CALL JOB:SEARCH-R1-S13D
SET P042 P006
SFTON3D P042
SMOVL C00207 BC00207 V=60.0  +MOVJ EC00207
SMOVL C00208 BC00208 V=60.0  +MOVJ EC00208
SREFP 3 C00209 BC00209  +REFP EC00209
CALL JOB:SEARCH-R1-S13D
SET P042 P006
SFTON3D P042
SMOVL C00210 BC00210 V=60.0  +MOVJ EC00210
MOVL C00211 BC00211 V=400.0  +MOVJ EC00211 VJ=100.00
MOVL C00212 BC00212 V=1000.0  +MOVJ EC00212 VJ=100.00
'Path S1165
SFTOF3D
MOVJ C00213 BC00213 VJ=100.00  +MOVJ EC00213 VJ=100.00
MOVL C00214 BC00214 V=400.0  +MOVJ EC00214 VJ=100.00
SMOVL C00215 BC00215 V=60.0  +MOVJ EC00215
SREFP 3 C00216 BC00216  +REFP EC00216
CALL JOB:SEARCH-R1-S13D
SET P041 P006
SFTON3D P041
SMOVL C00217 BC00217 V=60.0  +MOVJ EC00217
SMOVL C00218 BC00218 V=60.0  +MOVJ EC00218
SREFP 3 C00219 BC00219  +REFP EC00219
CALL JOB:SEARCH-R1-S13D
SET P041 P006
SFTON3D P041
SMOVL C00220 BC00220 V=60.0  +MOVJ EC00220
SMOVL C00221 BC00221 V=60.0  +MOVJ EC00221
SREFP 3 C00222 BC00222  +REFP EC00222
CALL JOB:SEARCH-R1-S13D
SET P041 P006
SFTON3D P041
SMOVL C00223 BC00223 V=60.0  +MOVJ EC00223
MOVL C00224 BC00224 V=400.0  +MOVJ EC00224 VJ=100.00
MOVL C00225 BC00225 V=1000.0  +MOVJ EC00225 VJ=100.00
'Path W378
SFTOF3D
SFTON3D P041
MOVJ C00226 BC00226 VJ=100.00  +MOVJ EC00226 VJ=100.00
SMOVL C00227 BC00227 V=400.0  +MOVJ EC00227
SMOVL C00228 BC00228 V=100.0 PL=0  +MOVJ EC00228
SREFP 1 C00229 BC00229  +REFP EC00229
SREFP 2 C00230 BC00230  +REFP EC00230
MACRO1 MJ#(0) ARGF0
ARCON
SMOVL C00231 BC00231 V=8.3  +MOVJ EC00231
SMOVL C00232 BC00232 V=10.0  +MOVJ EC00232
SMOVL C00233 BC00233 V=10.0  +MOVJ EC00233
ARCOF
SMOVL C00234 BC00234 V=400.0  +MOVJ EC00234
SMOVL C00235 BC00235 V=1000.0  +MOVJ EC00235
SFTOF3D
'Path W379
SFTOF3D
SFTON3D P042
MOVJ C00236 BC00236 VJ=100.00  +MOVJ EC00236 VJ=100.00
MOVJ C00237 BC00237 VJ=100.00  +MOVJ EC00237 VJ=100.00
SMOVL C00238 BC00238 V=400.0  +MOVJ EC00238
SMOVL C00239 BC00239 V=100.0 PL=0  +MOVJ EC00239
SREFP 1 C00240 BC00240  +REFP EC00240
SREFP 2 C00241 BC00241  +REFP EC00241
MACRO1 MJ#(0) ARGF0
ARCON
SMOVL C00242 BC00242 V=10.0  +MOVJ EC00242
SMOVL C00243 BC00243 V=10.0  +MOVJ EC00243
SMOVL C00244 BC00244 V=10.0  +MOVJ EC00244
ARCOF
SMOVL C00245 BC00245 V=400.0  +MOVJ EC00245
SMOVL C00246 BC00246 V=1000.0  +MOVJ EC00246
SFTOF3D
MOVJ C00247 BC00247 VJ=100.00  +MOVJ EC00247 VJ=100.00
'Path W380
SFTOF3D
SFTON3D P043
MOVJ C00248 BC00248 VJ=100.00  +MOVJ EC00248 VJ=100.00
MOVJ C00249 BC00249 VJ=100.00  +MOVJ EC00249 VJ=100.00
SMOVL C00250 BC00250 V=400.0  +MOVJ EC00250
SMOVL C00251 BC00251 V=100.0 PL=0  +MOVJ EC00251
SREFP 1 C00252 BC00252  +REFP EC00252
SREFP 2 C00253 BC00253  +REFP EC00253
MACRO1 MJ#(0) ARGF0
ARCON
SMOVL C00254 BC00254 V=10.0  +MOVJ EC00254
SMOVL C00255 BC00255 V=10.0  +MOVJ EC00255
SMOVL C00256 BC00256 V=10.0  +MOVJ EC00256
ARCOF
SMOVL C00257 BC00257 V=400.0  +MOVJ EC00257
SMOVL C00258 BC00258 V=1000.0  +MOVJ EC00258
SMOVL C00259 BC00259 V=1000.0  +MOVJ EC00259
SFTOF3D
'Path W381
SFTOF3D
SFTON3D P044
MOVJ C00260 BC00260 VJ=100.00  +MOVJ EC00260 VJ=100.00
COMM SMOVL C00261 BC00261 V=400.0  +MOVJ EC00261
COMM SMOVL C00262 BC00262 V=100.0 PL=0  +MOVJ EC00262
COMM SREFP 1 C00263 BC00263  +REFP EC00263
COMM SREFP 2 C00264 BC00264  +REFP EC00264
COMM MACRO1 MJ#(0) ARGF0
COMM ARCON
COMM SMOVL C00265 BC00265 V=10.0  +MOVJ EC00265
COMM SMOVL C00266 BC00266 V=10.0  +MOVJ EC00266
COMM SMOVL C00267 BC00267 V=10.0  +MOVJ EC00267
COMM SMOVL C00268 BC00268 V=10.0  +MOVJ EC00268
COMM SMOVL C00269 BC00269 V=10.0  +MOVJ EC00269
COMM SMOVL C00270 BC00270 V=10.0  +MOVJ EC00270
COMM SMOVL C00271 BC00271 V=10.0  +MOVJ EC00271
COMM SMOVL C00272 BC00272 V=10.0  +MOVJ EC00272
COMM SMOVL C00273 BC00273 V=10.0  +MOVJ EC00273
COMM SMOVL C00274 BC00274 V=10.0  +MOVJ EC00274
COMM SMOVL C00275 BC00275 V=10.0  +MOVJ EC00275
COMM SMOVL C00276 BC00276 V=10.0  +MOVJ EC00276
COMM SMOVL C00277 BC00277 V=10.0  +MOVJ EC00277
COMM SMOVL C00278 BC00278 V=10.0  +MOVJ EC00278
COMM SMOVL C00279 BC00279 V=10.0  +MOVJ EC00279
COMM SMOVL C00280 BC00280 V=10.0  +MOVJ EC00280
COMM SMOVL C00281 BC00281 V=10.0  +MOVJ EC00281
COMM SMOVL C00282 BC00282 V=10.0  +MOVJ EC00282
COMM SMOVL C00283 BC00283 V=10.0  +MOVJ EC00283
COMM SMOVL C00284 BC00284 V=10.0  +MOVJ EC00284
COMM SMOVL C00285 BC00285 V=10.0  +MOVJ EC00285
COMM SMOVL C00286 BC00286 V=10.0  +MOVJ EC00286
COMM SMOVL C00287 BC00287 V=10.0  +MOVJ EC00287
COMM SMOVL C00288 BC00288 V=10.0  +MOVJ EC00288
COMM SMOVL C00289 BC00289 V=10.0  +MOVJ EC00289
COMM ARCOF
COMM SMOVL C00290 BC00290 V=400.0  +MOVJ EC00290
SMOVL C00291 BC00291 V=1000.0  +MOVJ EC00291
SFTOF3D
'Path W382
SFTOF3D
SFTON3D P045
MOVJ C00292 BC00292 VJ=100.00  +MOVJ EC00292 VJ=100.00
SMOVL C00293 BC00293 V=400.0  +MOVJ EC00293
SMOVL C00294 BC00294 V=100.0 PL=0  +MOVJ EC00294
SREFP 1 C00295 BC00295  +REFP EC00295
SREFP 2 C00296 BC00296  +REFP EC00296
MACRO1 MJ#(0) ARGF0
ARCON
SMOVL C00297 BC00297 V=10.0  +MOVJ EC00297
SMOVL C00298 BC00298 V=10.0  +MOVJ EC00298
SMOVL C00299 BC00299 V=10.0  +MOVJ EC00299
ARCOF
SMOVL C00300 BC00300 V=400.0  +MOVJ EC00300
SMOVL C00301 BC00301 V=1000.0  +MOVJ EC00301
SMOVL C00302 BC00302 V=1000.0  +MOVJ EC00302
SFTOF3D
MOVJ C00303 BC00303 VJ=100.00  +MOVJ EC00303 VJ=100.00
'Path W383
SFTOF3D
SFTON3D P046
MOVJ C00304 BC00304 VJ=100.00  +MOVJ EC00304 VJ=100.00
MOVJ C00305 BC00305 VJ=100.00  +MOVJ EC00305 VJ=100.00
SMOVL C00306 BC00306 V=400.0  +MOVJ EC00306
SMOVL C00307 BC00307 V=100.0 PL=0  +MOVJ EC00307
SREFP 1 C00308 BC00308  +REFP EC00308
SREFP 2 C00309 BC00309  +REFP EC00309
MACRO1 MJ#(0) ARGF0
ARCON
SMOVL C00310 BC00310 V=10.0  +MOVJ EC00310
SMOVL C00311 BC00311 V=10.0  +MOVJ EC00311
SMOVL C00312 BC00312 V=10.0  +MOVJ EC00312
ARCOF
SMOVL C00313 BC00313 V=400.0  +MOVJ EC00313
SMOVL C00314 BC00314 V=1000.0  +MOVJ EC00314
SFTOF3D
MOVJ C00315 BC00315 VJ=100.00  +MOVJ EC00315 VJ=100.00
MOVJ C00316 BC00316 VJ=100.00  +MOVJ EC00316 VJ=100.00
'Down
MOVJ C00317 BC00317 VJ=100.00  +MOVJ EC00317 VJ=100.00
MOVJ C00318 BC00318 VJ=100.00  +MOVJ EC00318 VJ=100.00
COMM 'Path W1720
COMM SFTOF3D
COMM SFTON3D P032
COMM MOVJ C00319 BC00319 VJ=100.00  +MOVJ EC00319 VJ=100.00
COMM SMOVL C00320 BC00320 V=400.0  +MOVJ EC00320
COMM SMOVL C00321 BC00321 V=100.0 PL=0  +MOVJ EC00321
COMM SREFP 1 C00322 BC00322  +REFP EC00322
COMM SREFP 2 C00323 BC00323  +REFP EC00323
COMM MACRO1 MJ#(0) ARGF0
COMM ARCON
COMM SMOVL C00324 BC00324 V=10.0  +MOVJ EC00324
COMM SMOVL C00325 BC00325 V=10.0  +MOVJ EC00325
COMM SMOVL C00326 BC00326 V=10.0  +MOVJ EC00326
COMM SMOVL C00327 BC00327 V=10.0  +MOVJ EC00327
COMM SMOVL C00328 BC00328 V=10.0  +MOVJ EC00328
COMM SMOVL C00329 BC00329 V=10.0  +MOVJ EC00329
COMM SMOVL C00330 BC00330 V=10.0  +MOVJ EC00330
COMM SMOVL C00331 BC00331 V=10.0  +MOVJ EC00331
COMM SMOVL C00332 BC00332 V=10.0  +MOVJ EC00332
COMM SMOVL C00333 BC00333 V=10.0  +MOVJ EC00333
COMM SMOVL C00334 BC00334 V=10.0  +MOVJ EC00334
COMM SMOVL C00335 BC00335 V=10.0  +MOVJ EC00335
COMM SMOVL C00336 BC00336 V=10.0  +MOVJ EC00336
COMM SMOVL C00337 BC00337 V=10.0  +MOVJ EC00337
COMM SMOVL C00338 BC00338 V=10.0  +MOVJ EC00338
COMM ARCOF
COMM SMOVL C00339 BC00339 V=400.0  +MOVJ EC00339
COMM SMOVL C00340 BC00340 V=1000.0  +MOVJ EC00340
COMM SFTOF3D
COMM MOVJ C00341 BC00341 VJ=100.00  +MOVJ EC00341 VJ=100.00
MOVJ C00342 BC00342 VJ=100.00  +MOVJ EC00342 VJ=100.00
MOVJ C00343 BC00343 VJ=100.00  +MOVJ EC00343 VJ=100.00
MOVJ C00344 BC00344 VJ=100.00  +MOVJ EC00344 VJ=100.00
MOVJ C00345 BC00345 VJ=100.00  +MOVJ EC00345 VJ=100.00
'Path W1626
SFTOF3D
SFTON3D P022
MOVJ C00346 BC00346 VJ=100.00  +MOVJ EC00346 VJ=100.00
SMOVL C00347 BC00347 V=100.0  +MOVJ EC00347
SMOVL C00348 BC00348 V=100.0 PL=0  +MOVJ EC00348
SREFP 1 C00349 BC00349  +REFP EC00349
SREFP 2 C00350 BC00350  +REFP EC00350
MACRO1 MJ#(0) ARGF0
ARCON
SMOVC C00351 BC00351 V=11.0  +MOVJ EC00351
SMOVC C00352 BC00352 V=11.0  +MOVJ EC00352
SMOVC C00353 BC00353 V=11.0  +MOVJ EC00353
SMOVC C00354 BC00354 V=11.0  +MOVJ EC00354
ARCOF
SMOVL C00355 BC00355 V=400.0  +MOVJ EC00355
SMOVL C00356 BC00356 V=1000.0  +MOVJ EC00356
SFTOF3D
'Path W1627
SFTOF3D
SFTON3D P022
MOVJ C00357 BC00357 VJ=100.00  +MOVJ EC00357 VJ=100.00
SMOVL C00358 BC00358 V=100.0  +MOVJ EC00358
SMOVL C00359 BC00359 V=100.0 PL=0  +MOVJ EC00359
SREFP 1 C00360 BC00360  +REFP EC00360
SREFP 2 C00361 BC00361  +REFP EC00361
MACRO1 MJ#(0) ARGF0
ARCON
SMOVL C00362 BC00362 V=10.0  +MOVJ EC00362
SMOVL C00363 BC00363 V=10.0  +MOVJ EC00363
SMOVL C00364 BC00364 V=10.0  +MOVJ EC00364
ARCOF
SMOVL C00365 BC00365 V=400.0  +MOVJ EC00365
SMOVL C00366 BC00366 V=1000.0  +MOVJ EC00366
SFTOF3D
MOVJ C00367 BC00367 VJ=100.00  +MOVJ EC00367 VJ=100.00
'
'Path W1629
SFTOF3D
SFTON3D P023
MOVJ C00368 BC00368 VJ=100.00  +MOVJ EC00368 VJ=100.00
COMM MOVJ C00369 BC00369 VJ=100.00  +MOVJ EC00369 VJ=100.00
COMM SMOVL C00370 BC00370 V=400.0  +MOVJ EC00370
COMM SMOVL C00371 BC00371 V=100.0 PL=0  +MOVJ EC00371
COMM SREFP 1 C00372 BC00372  +REFP EC00372
COMM SREFP 2 C00373 BC00373  +REFP EC00373
COMM MACRO1 MJ#(0) ARGF0
COMM ARCON
COMM SMOVL C00374 BC00374 V=10.0  +MOVJ EC00374
COMM SMOVL C00375 BC00375 V=10.0  +MOVJ EC00375
COMM SMOVL C00376 BC00376 V=10.0  +MOVJ EC00376
COMM ARCOF
COMM SMOVL C00377 BC00377 V=400.0  +MOVJ EC00377
COMM SMOVL C00378 BC00378 V=1000.0  +MOVJ EC00378
COMM SFTOF3D
COMM 'Path W1630
COMM SFTOF3D
COMM SFTON3D P023
COMM MOVJ C00379 BC00379 VJ=100.00  +MOVJ EC00379 VJ=100.00
COMM SMOVL C00380 BC00380 V=100.0  +MOVJ EC00380
COMM SMOVL C00381 BC00381 V=100.0 PL=0  +MOVJ EC00381
COMM SREFP 1 C00382 BC00382  +REFP EC00382
COMM SREFP 2 C00383 BC00383  +REFP EC00383
COMM MACRO1 MJ#(0) ARGF0
COMM ARCON
COMM SMOVL C00384 BC00384 V=10.0  +MOVJ EC00384
COMM SMOVL C00385 BC00385 V=10.0  +MOVJ EC00385
COMM SMOVL C00386 BC00386 V=10.0  +MOVJ EC00386
COMM ARCOF
COMM SMOVL C00387 BC00387 V=400.0  +MOVJ EC00387
COMM SMOVL C00388 BC00388 V=1000.0  +MOVJ EC00388
COMM SMOVL C00389 BC00389 V=1000.0  +MOVJ EC00389
COMM SFTOF3D
COMM 'Path W1631
COMM SFTOF3D
COMM SFTON3D P023
COMM MOVJ C00390 BC00390 VJ=100.00  +MOVJ EC00390 VJ=100.00
COMM SMOVL C00391 BC00391 V=100.0  +MOVJ EC00391
COMM SMOVL C00392 BC00392 V=100.0 PL=0  +MOVJ EC00392
COMM SREFP 1 C00393 BC00393  +REFP EC00393
COMM SREFP 2 C00394 BC00394  +REFP EC00394
COMM MACRO1 MJ#(0) ARGF0
COMM ARCON
COMM SMOVL C00395 BC00395 V=10.0  +MOVJ EC00395
COMM ARCOF
COMM SMOVL C00396 BC00396 V=400.0  +MOVJ EC00396
COMM SMOVL C00397 BC00397 V=1000.0  +MOVJ EC00397
COMM SFTOF3D
COMM '
COMM 'Path W1632
COMM SFTOF3D
COMM SFTON3D P024
COMM MOVJ C00398 BC00398 VJ=100.00  +MOVJ EC00398 VJ=100.00
COMM SMOVL C00399 BC00399 V=100.0  +MOVJ EC00399
COMM SMOVL C00400 BC00400 V=100.0 PL=0  +MOVJ EC00400
COMM SREFP 1 C00401 BC00401  +REFP EC00401
COMM SREFP 2 C00402 BC00402  +REFP EC00402
COMM MACRO1 MJ#(0) ARGF0
COMM ARCON
COMM SMOVL C00403 BC00403 V=10.0  +MOVJ EC00403
COMM SMOVL C00404 BC00404 V=10.0  +MOVJ EC00404
COMM SMOVL C00405 BC00405 V=10.0  +MOVJ EC00405
COMM ARCOF
COMM SMOVL C00406 BC00406 V=400.0  +MOVJ EC00406
COMM SMOVL C00407 BC00407 V=1000.0  +MOVJ EC00407
COMM SFTOF3D
COMM 'Path W1633
COMM SFTOF3D
COMM SFTON3D P024
COMM MOVJ C00408 BC00408 VJ=100.00  +MOVJ EC00408 VJ=100.00
COMM SMOVL C00409 BC00409 V=100.0  +MOVJ EC00409
COMM SMOVL C00410 BC00410 V=100.0 PL=0  +MOVJ EC00410
COMM SREFP 1 C00411 BC00411  +REFP EC00411
COMM SREFP 2 C00412 BC00412  +REFP EC00412
COMM MACRO1 MJ#(0) ARGF0
COMM ARCON
COMM SMOVL C00413 BC00413 V=10.0  +MOVJ EC00413
COMM SMOVL C00414 BC00414 V=10.0  +MOVJ EC00414
COMM SMOVL C00415 BC00415 V=10.0  +MOVJ EC00415
COMM ARCOF
COMM SMOVL C00416 BC00416 V=400.0  +MOVJ EC00416
COMM SMOVL C00417 BC00417 V=1000.0  +MOVJ EC00417
COMM SMOVL C00418 BC00418 V=1000.0  +MOVJ EC00418
COMM SFTOF3D
COMM 'Path W1634
COMM SFTOF3D
COMM SFTON3D P024
COMM MOVJ C00419 BC00419 VJ=100.00  +MOVJ EC00419 VJ=100.00
COMM SMOVL C00420 BC00420 V=100.0  +MOVJ EC00420
COMM SMOVL C00421 BC00421 V=100.0 PL=0  +MOVJ EC00421
COMM SREFP 1 C00422 BC00422  +REFP EC00422
COMM SREFP 2 C00423 BC00423  +REFP EC00423
COMM MACRO1 MJ#(0) ARGF0
COMM ARCON
COMM SMOVL C00424 BC00424 V=10.0  +MOVJ EC00424
COMM ARCOF
COMM SMOVL C00425 BC00425 V=400.0  +MOVJ EC00425
COMM SMOVL C00426 BC00426 V=1000.0  +MOVJ EC00426
COMM SFTOF3D
COMM '
COMM 'Path W1635
COMM SFTOF3D
COMM SFTON3D P025
COMM MOVJ C00427 BC00427 VJ=100.00  +MOVJ EC00427 VJ=100.00
COMM SMOVL C00428 BC00428 V=100.0  +MOVJ EC00428
COMM SMOVL C00429 BC00429 V=100.0 PL=0  +MOVJ EC00429
COMM SREFP 1 C00430 BC00430  +REFP EC00430
COMM SREFP 2 C00431 BC00431  +REFP EC00431
COMM MACRO1 MJ#(0) ARGF0
COMM ARCON
COMM SMOVL C00432 BC00432 V=10.0  +MOVJ EC00432
COMM SMOVL C00433 BC00433 V=10.0  +MOVJ EC00433
COMM SMOVL C00434 BC00434 V=10.0  +MOVJ EC00434
COMM ARCOF
COMM SMOVL C00435 BC00435 V=400.0  +MOVJ EC00435
COMM SMOVL C00436 BC00436 V=1000.0  +MOVJ EC00436
COMM SFTOF3D
COMM 'Path W1636
COMM SFTOF3D
COMM SFTON3D P025
COMM MOVJ C00437 BC00437 VJ=100.00  +MOVJ EC00437 VJ=100.00
COMM SMOVL C00438 BC00438 V=100.0  +MOVJ EC00438
COMM SMOVL C00439 BC00439 V=100.0 PL=0  +MOVJ EC00439
COMM SREFP 1 C00440 BC00440  +REFP EC00440
COMM SREFP 2 C00441 BC00441  +REFP EC00441
COMM MACRO1 MJ#(0) ARGF0
COMM ARCON
COMM SMOVL C00442 BC00442 V=10.0  +MOVJ EC00442
COMM SMOVL C00443 BC00443 V=10.0  +MOVJ EC00443
COMM SMOVL C00444 BC00444 V=10.0  +MOVJ EC00444
COMM ARCOF
COMM SMOVL C00445 BC00445 V=400.0  +MOVJ EC00445
COMM SMOVL C00446 BC00446 V=1000.0  +MOVJ EC00446
COMM SMOVL C00447 BC00447 V=1000.0  +MOVJ EC00447
COMM SFTOF3D
COMM 'Path W1637
COMM SFTOF3D
COMM SFTON3D P025
COMM MOVJ C00448 BC00448 VJ=100.00  +MOVJ EC00448 VJ=100.00
COMM SMOVL C00449 BC00449 V=100.0  +MOVJ EC00449
COMM SMOVL C00450 BC00450 V=100.0 PL=0  +MOVJ EC00450
COMM SREFP 1 C00451 BC00451  +REFP EC00451
COMM SREFP 2 C00452 BC00452  +REFP EC00452
COMM MACRO1 MJ#(0) ARGF0
COMM ARCON
COMM SMOVL C00453 BC00453 V=10.0  +MOVJ EC00453
COMM ARCOF
COMM SMOVL C00454 BC00454 V=400.0  +MOVJ EC00454
COMM SMOVL C00455 BC00455 V=1000.0  +MOVJ EC00455
COMM SFTOF3D
COMM MOVJ C00456 BC00456 VJ=100.00  +MOVJ EC00456 VJ=100.00
COMM MOVJ C00457 BC00457 VJ=100.00  +MOVJ EC00457 VJ=100.00
COMM MOVJ C00458 BC00458 VJ=100.00  +MOVJ EC00458 VJ=100.00
COMM '
COMM 'Path W1639
COMM SFTOF3D
COMM SFTON3D P023
COMM SMOVL C00459 BC00459 V=100.0  +MOVJ EC00459
COMM SMOVL C00460 BC00460 V=100.0 PL=0  +MOVJ EC00460
COMM SREFP 1 C00461 BC00461  +REFP EC00461
COMM SREFP 2 C00462 BC00462  +REFP EC00462
COMM MACRO1 MJ#(0) ARGF0
COMM ARCON
COMM SMOVL C00463 BC00463 V=10.0  +MOVJ EC00463
COMM SMOVL C00464 BC00464 V=10.0  +MOVJ EC00464
COMM SMOVL C00465 BC00465 V=10.0  +MOVJ EC00465
COMM ARCOF
COMM SMOVL C00466 BC00466 V=400.0  +MOVJ EC00466
COMM SFTOF3D
COMM 'Path W1638
COMM SFTOF3D
COMM SFTON3D P023
COMM SMOVL C00467 BC00467 V=100.0  +MOVJ EC00467
COMM SMOVL C00468 BC00468 V=100.0 PL=0  +MOVJ EC00468
COMM SREFP 1 C00469 BC00469  +REFP EC00469
COMM SREFP 2 C00470 BC00470  +REFP EC00470
COMM MACRO1 MJ#(0) ARGF0
COMM ARCON
COMM SMOVL C00471 BC00471 V=10.0  +MOVJ EC00471
COMM SMOVL C00472 BC00472 V=10.0  +MOVJ EC00472
COMM SMOVL C00473 BC00473 V=10.0  +MOVJ EC00473
COMM ARCOF
COMM SMOVL C00474 BC00474 V=400.0  +MOVJ EC00474
COMM SFTOF3D
COMM MOVJ C00475 BC00475 VJ=100.00  +MOVJ EC00475 VJ=100.00
COMM '
COMM 'Path W1640
COMM SFTOF3D
COMM SFTON3D P024
COMM MOVJ C00476 BC00476 VJ=100.00  +MOVJ EC00476 VJ=100.00
COMM MOVJ C00477 BC00477 VJ=100.00  +MOVJ EC00477 VJ=100.00
COMM SMOVL C00478 BC00478 V=400.0  +MOVJ EC00478
COMM SMOVL C00479 BC00479 V=100.0 PL=0  +MOVJ EC00479
COMM SREFP 1 C00480 BC00480  +REFP EC00480
COMM SREFP 2 C00481 BC00481  +REFP EC00481
COMM MACRO1 MJ#(0) ARGF0
COMM ARCON
COMM SMOVL C00482 BC00482 V=10.0  +MOVJ EC00482
COMM SMOVL C00483 BC00483 V=10.0  +MOVJ EC00483
COMM SMOVL C00484 BC00484 V=10.0  +MOVJ EC00484
COMM ARCOF
COMM SMOVL C00485 BC00485 V=400.0  +MOVJ EC00485
COMM SMOVL C00486 BC00486 V=1000.0  +MOVJ EC00486
COMM SMOVL C00487 BC00487 V=1000.0  +MOVJ EC00487
COMM SFTOF3D
COMM 'Path W1641
COMM SFTOF3D
COMM SFTON3D P025
COMM SMOVL C00488 BC00488 V=100.0  +MOVJ EC00488
COMM SMOVL C00489 BC00489 V=100.0 PL=0  +MOVJ EC00489
COMM SREFP 1 C00490 BC00490  +REFP EC00490
COMM SREFP 2 C00491 BC00491  +REFP EC00491
COMM MACRO1 MJ#(0) ARGF0
COMM ARCON
COMM SMOVL C00492 BC00492 V=10.0  +MOVJ EC00492
COMM SMOVL C00493 BC00493 V=10.0  +MOVJ EC00493
COMM SMOVL C00494 BC00494 V=10.0  +MOVJ EC00494
COMM ARCOF
COMM SMOVL C00495 BC00495 V=400.0  +MOVJ EC00495
COMM SMOVL C00496 BC00496 V=1000.0  +MOVJ EC00496
COMM SMOVL C00497 BC00497 V=1000.0  +MOVJ EC00497
COMM SFTOF3D
COMM MOVJ C00498 BC00498 VJ=100.00  +MOVJ EC00498 VJ=100.00
'DO USUNIECIA
'DO USUNIECIA
MOVL C00499 BC00499 V=83.3  +MOVJ EC00499 VJ=0.78
MOVL C00500 BC00500 V=83.3  +MOVJ EC00500 VJ=0.78
MOVL C00501 BC00501 V=83.3  +MOVJ EC00501 VJ=0.78
MOVL C00502 BC00502 V=83.3  +MOVJ EC00502 VJ=0.78
'DO USUNIECIA
'DO USUNIECIA
MOVJ C00503 BC00503 VJ=100.00  +MOVJ EC00503 VJ=100.00
MOVJ C00504 BC00504 VJ=100.00  +MOVJ EC00504 VJ=100.00
MOVJ C00505 BC00505 VJ=100.00  +MOVJ EC00505 VJ=100.00
'Path W1911
SFTOF3D
SFTON3D P021
MOVJ C00506 BC00506 VJ=100.00  +MOVJ EC00506 VJ=100.00
SMOVL C00507 BC00507 V=100.0  +MOVJ EC00507
SMOVL C00508 BC00508 V=100.0 PL=0  +MOVJ EC00508
SREFP 1 C00509 BC00509  +REFP EC00509
SREFP 2 C00510 BC00510  +REFP EC00510
MACRO1 MJ#(0) ARGF0
ARCON
SMOVC C00511 BC00511 V=10.0  +MOVJ EC00511
SMOVC C00512 BC00512 V=10.0  +MOVJ EC00512
SMOVC C00513 BC00513 V=10.0  +MOVJ EC00513
SMOVC C00514 BC00514 V=10.0  +MOVJ EC00514
ARCOF
SMOVL C00515 BC00515 V=400.0  +MOVJ EC00515
SMOVL C00516 BC00516 V=1000.0  +MOVJ EC00516
SFTOF3D
MOVJ C00517 BC00517 VJ=100.00  +MOVJ EC00517 VJ=100.00
MOVJ C00518 BC00518 VJ=100.00  +MOVJ EC00518 VJ=100.00
'
MOVJ C00519 BC00519 VJ=100.00  +MOVJ EC00519 VJ=100.00
COMM MOVJ C00520 BC00520 VJ=100.00  +MOVJ EC00520 VJ=100.00
COMM 'Path W1642
COMM SFTOF3D
COMM SFTON3D P024
COMM MOVJ C00521 BC00521 VJ=100.00  +MOVJ EC00521 VJ=100.00
COMM SMOVL C00522 BC00522 V=100.0  +MOVJ EC00522
COMM SMOVL C00523 BC00523 V=100.0 PL=0  +MOVJ EC00523
COMM SREFP 1 C00524 BC00524  +REFP EC00524
COMM SREFP 2 C00525 BC00525  +REFP EC00525
COMM MACRO1 MJ#(0) ARGF0
COMM ARCON
COMM SMOVL C00526 BC00526 V=10.0  +MOVJ EC00526
COMM SMOVL C00527 BC00527 V=10.0  +MOVJ EC00527
COMM SMOVL C00528 BC00528 V=10.0  +MOVJ EC00528
COMM ARCOF
COMM SMOVL C00529 BC00529 V=400.0  +MOVJ EC00529
COMM SMOVL C00530 BC00530 V=1000.0  +MOVJ EC00530
COMM SFTOF3D
COMM 'Path W1643
SFTOF3D
SFTON3D P025
COMM MOVJ C00531 BC00531 VJ=100.00  +MOVJ EC00531 VJ=100.00
COMM SMOVL C00532 BC00532 V=100.0  +MOVJ EC00532
COMM SMOVL C00533 BC00533 V=100.0 PL=0  +MOVJ EC00533
COMM SREFP 1 C00534 BC00534  +REFP EC00534
COMM SREFP 2 C00535 BC00535  +REFP EC00535
COMM MACRO1 MJ#(0) ARGF0
COMM ARCON
COMM SMOVL C00536 BC00536 V=10.0  +MOVJ EC00536
COMM SMOVL C00537 BC00537 V=10.0  +MOVJ EC00537
COMM SMOVL C00538 BC00538 V=10.0  +MOVJ EC00538
COMM ARCOF
COMM SMOVL C00539 BC00539 V=400.0  +MOVJ EC00539
COMM SMOVL C00540 BC00540 V=1000.0  +MOVJ EC00540
COMM SMOVL C00541 BC00541 V=1000.0  +MOVJ EC00541
COMM SFTOF3D
COMM '
COMM 'Path W1644
SFTOF3D
SFTON3D P026
MOVJ C00542 BC00542 VJ=50.00  +MOVJ EC00542 VJ=50.00
MOVJ C00543 BC00543 VJ=100.00  +MOVJ EC00543 VJ=100.00
SMOVL C00544 BC00544 V=100.0  +MOVJ EC00544
SMOVL C00545 BC00545 V=100.0 PL=0  +MOVJ EC00545
SREFP 1 C00546 BC00546  +REFP EC00546
SREFP 2 C00547 BC00547  +REFP EC00547
MACRO1 MJ#(0) ARGF0
ARCON
SMOVC C00548 BC00548 V=10.0  +MOVJ EC00548
SMOVC C00549 BC00549 V=10.0  +MOVJ EC00549
SMOVC C00550 BC00550 V=10.0  +MOVJ EC00550
ARCOF
SMOVL C00551 BC00551 V=400.0  +MOVJ EC00551
SMOVL C00552 BC00552 V=1000.0  +MOVJ EC00552
SFTOF3D
'Path W1645
SFTOF3D
SFTON3D P027
MOVJ C00553 BC00553 VJ=100.00  +MOVJ EC00553 VJ=100.00
SMOVL C00554 BC00554 V=100.0  +MOVJ EC00554
SMOVL C00555 BC00555 V=100.0 PL=0  +MOVJ EC00555
SREFP 1 C00556 BC00556  +REFP EC00556
SREFP 2 C00557 BC00557  +REFP EC00557
MACRO1 MJ#(0) ARGF0
ARCON
SMOVL C00558 BC00558 V=10.0  +MOVJ EC00558
ARCOF
SMOVL C00559 BC00559 V=400.0  +MOVJ EC00559
SMOVL C00560 BC00560 V=1000.0  +MOVJ EC00560
SFTOF3D
MOVJ C00561 BC00561 VJ=100.00  +MOVJ EC00561 VJ=100.00
MOVJ C00562 BC00562 VJ=100.00  +MOVJ EC00562 VJ=100.00
'jakie searche do takicj spoin?
MOVJ C00563 BC00563 VJ=100.00  +MOVJ EC00563 VJ=100.00
'Path W1646
SFTOF3D
MOVJ C00564 BC00564 VJ=100.00  +MOVJ EC00564 VJ=100.00
MOVL C00565 BC00565 V=100.0  +MOVJ EC00565 VJ=100.00
SMOVL C00566 BC00566 V=100.0 PL=0  +MOVJ EC00566
SREFP 1 C00567 BC00567  +REFP EC00567
SREFP 2 C00568 BC00568  +REFP EC00568
MACRO1 MJ#(0) ARGF0
ARCON
SMOVL C00569 BC00569 V=10.0  +MOVJ EC00569
ARCOF
MOVL C00570 BC00570 V=400.0  +MOVJ EC00570 VJ=100.00
MOVL C00571 BC00571 V=1000.0  +MOVJ EC00571 VJ=100.00
MOVL C00572 BC00572 V=1000.0  +MOVJ EC00572 VJ=100.00
MOVJ C00573 BC00573 VJ=100.00  +MOVJ EC00573 VJ=100.00
'brak dostÄpu do jednej spoiny
'Path W1647
SFTOF3D
MOVJ C00574 BC00574 VJ=100.00  +MOVJ EC00574 VJ=100.00
MOVJ C00575 BC00575 VJ=100.00  +MOVJ EC00575 VJ=100.00
MOVL C00576 BC00576 V=400.0  +MOVJ EC00576 VJ=100.00
SMOVL C00577 BC00577 V=100.0 PL=0  +MOVJ EC00577
SREFP 1 C00578 BC00578  +REFP EC00578
SREFP 2 C00579 BC00579  +REFP EC00579
MACRO1 MJ#(0) ARGF0
ARCON
SMOVL C00580 BC00580 V=10.0  +MOVJ EC00580
ARCOF
MOVL C00581 BC00581 V=400.0  +MOVJ EC00581 VJ=100.00
MOVL C00582 BC00582 V=1000.0  +MOVJ EC00582 VJ=100.00
'Path W1648
SFTOF3D
MOVJ C00583 BC00583 VJ=100.00  +MOVJ EC00583 VJ=100.00
MOVL C00584 BC00584 V=100.0  +MOVJ EC00584 VJ=100.00
SMOVL C00585 BC00585 V=100.0 PL=0  +MOVJ EC00585
SREFP 1 C00586 BC00586  +REFP EC00586
SREFP 2 C00587 BC00587  +REFP EC00587
MACRO1 MJ#(0) ARGF0
ARCON
SMOVL C00588 BC00588 V=10.0  +MOVJ EC00588
ARCOF
MOVL C00589 BC00589 V=400.0  +MOVJ EC00589 VJ=100.00
MOVL C00590 BC00590 V=1000.0  +MOVJ EC00590 VJ=100.00
MOVL C00591 BC00591 V=1000.0  +MOVJ EC00591 VJ=100.00
MOVL C00592 BC00592 V=333.3  +MOVJ EC00592 VJ=100.00
'Path W1649
SFTOF3D
MOVL C00593 BC00593 V=333.3  +MOVJ EC00593 VJ=50.00
MOVL C00594 BC00594 V=333.3  +MOVJ EC00594 VJ=100.00
MOVL C00595 BC00595 V=100.0  +MOVJ EC00595 VJ=100.00
SMOVL C00596 BC00596 V=100.0 PL=0  +MOVJ EC00596
SREFP 1 C00597 BC00597  +REFP EC00597
SREFP 2 C00598 BC00598  +REFP EC00598
MACRO1 MJ#(0) ARGF0
ARCON
SMOVL C00599 BC00599 V=10.0  +MOVJ EC00599
ARCOF
MOVL C00600 BC00600 V=400.0  +MOVJ EC00600 VJ=100.00
MOVL C00601 BC00601 V=1000.0  +MOVJ EC00601 VJ=100.00
'Path W1650
SFTOF3D
MOVJ C00602 BC00602 VJ=100.00  +MOVJ EC00602 VJ=100.00
MOVL C00603 BC00603 V=100.0  +MOVJ EC00603 VJ=100.00
SMOVL C00604 BC00604 V=100.0 PL=0  +MOVJ EC00604
SREFP 1 C00605 BC00605  +REFP EC00605
SREFP 2 C00606 BC00606  +REFP EC00606
MACRO1 MJ#(0) ARGF0
ARCON
SMOVL C00607 BC00607 V=10.0  +MOVJ EC00607
ARCOF
MOVL C00608 BC00608 V=400.0  +MOVJ EC00608 VJ=100.00
MOVL C00609 BC00609 V=1000.0  +MOVJ EC00609 VJ=100.00
'Path W1651
SFTOF3D
MOVJ C00610 BC00610 VJ=100.00  +MOVJ EC00610 VJ=100.00
MOVL C00611 BC00611 V=100.0  +MOVJ EC00611 VJ=100.00
SMOVL C00612 BC00612 V=100.0 PL=0  +MOVJ EC00612
SREFP 1 C00613 BC00613  +REFP EC00613
SREFP 2 C00614 BC00614  +REFP EC00614
MACRO1 MJ#(0) ARGF0
ARCON
SMOVL C00615 BC00615 V=10.0  +MOVJ EC00615
ARCOF
MOVL C00616 BC00616 V=400.0  +MOVJ EC00616 VJ=100.00
MOVL C00617 BC00617 V=1000.0  +MOVJ EC00617 VJ=100.00
'Path W1652
SFTOF3D
MOVJ C00618 BC00618 VJ=100.00  +MOVJ EC00618 VJ=100.00
MOVL C00619 BC00619 V=100.0  +MOVJ EC00619 VJ=100.00
SMOVL C00620 BC00620 V=100.0 PL=0  +MOVJ EC00620
SREFP 1 C00621 BC00621  +REFP EC00621
SREFP 2 C00622 BC00622  +REFP EC00622
MACRO1 MJ#(0) ARGF0
ARCON
SMOVL C00623 BC00623 V=10.0  +MOVJ EC00623
ARCOF
MOVL C00624 BC00624 V=400.0  +MOVJ EC00624 VJ=100.00
MOVL C00625 BC00625 V=1000.0  +MOVJ EC00625 VJ=100.00
'jakie searche do takicj spoin?
MOVJ C00626 BC00626 VJ=100.00  +MOVJ EC00626 VJ=100.00
'Path W1653
SFTOF3D
MOVJ C00627 BC00627 VJ=100.00  +MOVJ EC00627 VJ=100.00
MOVL C00628 BC00628 V=100.0  +MOVJ EC00628 VJ=100.00
SMOVL C00629 BC00629 V=100.0 PL=0  +MOVJ EC00629
SREFP 1 C00630 BC00630  +REFP EC00630
SREFP 2 C00631 BC00631  +REFP EC00631
MACRO1 MJ#(0) ARGF0
ARCON
SMOVL C00632 BC00632 V=10.0  +MOVJ EC00632
SMOVL C00633 BC00633 V=10.0  +MOVJ EC00633
ARCOF
MOVL C00634 BC00634 V=400.0  +MOVJ EC00634 VJ=100.00
MOVL C00635 BC00635 V=1000.0  +MOVJ EC00635 VJ=100.00
MOVL C00636 BC00636 V=1000.0  +MOVJ EC00636 VJ=100.00
'Path W1654
SFTOF3D
MOVJ C00637 BC00637 VJ=100.00  +MOVJ EC00637 VJ=100.00
MOVL C00638 BC00638 V=100.0  +MOVJ EC00638 VJ=100.00
SMOVL C00639 BC00639 V=100.0 PL=0  +MOVJ EC00639
SREFP 1 C00640 BC00640  +REFP EC00640
